LIN {X 0,Y 185.602,Z 322.354,A -85,B 0,C 180,E1 -22115.385,E2 -22115.385} C_VEL
LIN {X 0,Y 185.671,Z 322.353,A -85,B 0,C 180,E1 -22121.133,E2 -22121.133} C_VEL
LIN {X 0,Y 185.762,Z 322.338,A -85,B 0,C 180,E1 -22126.88,E2 -22126.88} C_VEL
LIN {X 0,Y 186.021,Z 322.304,A -85,B 0,C 180,E1 -22131.308,E2 -22131.308} C_VEL
LIN {X 0,Y 186.205,Z 322.287,A -85,B 0,C 180,E1 -22137.837,E2 -22137.837} C_VEL
LIN {X 0,Y 186.404,Z 322.255,A -85,B 0,C 180,E1 -22140.001,E2 -22140.001} C_VEL
LIN {X 0,Y 185.924,Z 322.314,A -85,B 0,C 180,E1 -22144.336,E2 -22144.336} C_VEL
LIN {X 0,Y 186.026,Z 322.301,A -85,B 0,C 180,E1 -22148.692,E2 -22148.692} C_VEL
LIN {X 0,Y 185.762,Z 322.334,A -85,B 0,C 180,E1 -22153.121,E2 -22153.121} C_VEL
LIN {X 0,Y 185.714,Z 322.341,A -85,B 0,C 180,E1 -22157.623,E2 -22157.623} C_VEL
LIN {X 0,Y 185.631,Z 322.481,A -85,B 0,C 180,E1 -22163.056,E2 -22163.056} C_VEL
LIN {X 0,Y 186.574,Z 325.065,A -85,B 0,C 180,E1 -22163.814,E2 -22163.814} C_VEL
LIN {X 0,Y 188.555,Z 327.314,A -85,B 0,C 180,E1 -22165.085,E2 -22165.085} C_VEL
LIN {X 0,Y 189.992,Z 328.26,A -85,B 0,C 180,E1 -22165.911,E2 -22165.911} C_VEL
LIN {X 0,Y 191.804,Z 331.332,A -85,B 0,C 180,E1 -22167.039,E2 -22167.039} C_VEL
LIN {X 0,Y 194.147,Z 333.688,A -85,B 0,C 180,E1 -22168.307,E2 -22168.307} C_VEL
LIN {X 0,Y 196.773,Z 337.354,A -85,B 0,C 180,E1 -22169.708,E2 -22169.708} C_VEL
LIN {X 0,Y 197.995,Z 338.775,A -85,B 0,C 180,E1 -22170.313,E2 -22170.313} C_VEL
LIN {X 0,Y 200.923,Z 342.622,A -85,B 0,C 180,E1 -22171.724,E2 -22171.724} C_VEL
LIN {X 0,Y 207.739,Z 352.452,A -85,B 0,C 180,E1 -22174.74,E2 -22174.74} C_VEL
LIN {X 0,Y 214.156,Z 362.539,A -85,B 0,C 180,E1 -22177.29,E2 -22177.29} C_VEL
LIN {X 0,Y 221.381,Z 375.322,A -85,B 0,C 180,E1 -22179.914,E2 -22179.914} C_VEL
LIN {X 0,Y 223.449,Z 379.739,A -85,B 0,C 180,E1 -22180.645,E2 -22180.645} C_VEL
LIN {X 0,Y 220.676,Z 423.154,A -85,B 0,C 180,E1 -22181.949,E2 -22181.949} C_VEL
LIN {X 0,Y 219.117,Z 436.689,A -85,B 0,C 180,E1 -22182.72,E2 -22182.72} C_VEL
LIN {X 0,Y 216.946,Z 448.789,A -85,B 0,C 180,E1 -22183.714,E2 -22183.714} C_VEL
LIN {X 0,Y 213.831,Z 460.908,A -85,B 0,C 180,E1 -22185.039,E2 -22185.039} C_VEL
LIN {X 0,Y 210.401,Z 472.488,A -85,B 0,C 180,E1 -22186.785,E2 -22186.785} C_VEL
LIN {X 0,Y 207.063,Z 482.377,A -85,B 0,C 180,E1 -22188.73,E2 -22188.73} C_VEL
LIN {X 0,Y 203.419,Z 491.299,A -85,B 0,C 180,E1 -22190.913,E2 -22190.913} C_VEL
LIN {X 0,Y 199.211,Z 500.425,A -85,B 0,C 180,E1 -22193.787,E2 -22193.787} C_VEL
LIN {X 0,Y 195.528,Z 507.705,A -85,B 0,C 180,E1 -22196.762,E2 -22196.762} C_VEL
LIN {X 0,Y 192.756,Z 512.596,A -85,B 0,C 180,E1 -22199.308,E2 -22199.308} C_VEL
LIN {X 0,Y 189.694,Z 517.737,A -85,B 0,C 180,E1 -22202.772,E2 -22202.772} C_VEL
LIN {X 0,Y 187.644,Z 520.887,A -85,B 0,C 180,E1 -22205.671,E2 -22205.671} C_VEL
LIN {X 0,Y 186.386,Z 522.696,A -85,B 0,C 180,E1 -22207.849,E2 -22207.849} C_VEL
LIN {X 0,Y 184.582,Z 524.972,A -85,B 0,C 180,E1 -22212.267,E2 -22212.267} C_VEL
LIN {X 0,Y 183.944,Z 525.517,A -85,B 0,C 180,E1 -22214.489,E2 -22214.489} C_VEL
LIN {X 0,Y 183.457,Z 525.636,A -85,B 0,C 180,E1 -22216.713,E2 -22216.713} C_VEL
LIN {X 0,Y 183.163,Z 524.659,A -85,B 0,C 180,E1 -22221.173,E2 -22221.173} C_VEL
LIN {X 0,Y 183.461,Z 522.612,A -85,B 0,C 180,E1 -22224.887,E2 -22224.887} C_VEL
LIN {X 0,Y 183.924,Z 519.046,A -85,B 0,C 180,E1 -22228.907,E2 -22228.907} C_VEL
LIN {X 0,Y 184.855,Z 514.96,A -85,B 0,C 180,E1 -22232.18,E2 -22232.18} C_VEL
LIN {X 0,Y 186.297,Z 508.724,A -85,B 0,C 180,E1 -22235.956,E2 -22235.956} C_VEL
LIN {X 0,Y 188.111,Z 501.932,A -85,B 0,C 180,E1 -22239.138,E2 -22239.138} C_VEL
LIN {X 0,Y 190.326,Z 493.47,A -85,B 0,C 180,E1 -22242.26,E2 -22242.26} C_VEL
LIN {X 0,Y 192.574,Z 484.767,A -85,B 0,C 180,E1 -22244.802,E2 -22244.802} C_VEL
LIN {X 0,Y 195.141,Z 474.056,A -85,B 0,C 180,E1 -22247.286,E2 -22247.286} C_VEL
LIN {X 0,Y 197.445,Z 463.339,A -85,B 0,C 180,E1 -22249.225,E2 -22249.225} C_VEL
LIN {X 0,Y 199.409,Z 451.373,A -85,B 0,C 180,E1 -22250.908,E2 -22250.908} C_VEL
LIN {X 0,Y 201.104,Z 438.875,A -85,B 0,C 180,E1 -22252.203,E2 -22252.203} C_VEL
LIN {X 0,Y 202.264,Z 426.146,A -85,B 0,C 180,E1 -22253.12,E2 -22253.12} C_VEL
LIN {X 0,Y 203.098,Z 410.38,A -85,B 0,C 180,E1 -22253.767,E2 -22253.767} C_VEL
LIN {X 0,Y 205.254,Z 361.08,A -85,B 0,C 180,E1 -22255.386,E2 -22255.386} C_VEL
LIN {X 0,Y 198.748,Z 346.766,A -85,B 0,C 180,E1 -22257.112,E2 -22257.112} C_VEL
LIN {X 0,Y 191.698,Z 333.496,A -85,B 0,C 180,E1 -22259.053,E2 -22259.053} C_VEL
LIN {X 0,Y 187.267,Z 326.204,A -85,B 0,C 180,E1 -22260.324,E2 -22260.324} C_VEL
LIN {X 0,Y 185.864,Z 323.755,A -85,B 0,C 180,E1 -22260.749,E2 -22260.749} C_VEL
LIN {X 0,Y 185.524,Z 322.374,A -85,B 0,C 180,E1 -22260.905,E2 -22260.905} C_VEL
LIN {X 0,Y 185.502,Z 322.377,A -85,B 0,C 180,E1 -22264.633,E2 -22264.633} C_VEL
LIN {X 0,Y 185.504,Z 322.377,A -85,B 0,C 180,E1 -22267.315,E2 -22267.315} C_VEL
LIN {X 0,Y 185.466,Z 322.369,A -85,B 0,C 180,E1 -22270.722,E2 -22270.722} C_VEL
LIN {X 0,Y 185.46,Z 322.373,A -85,B 0,C 180,E1 -22276.057,E2 -22276.057} C_VEL
LIN {X 0,Y 185.46,Z 322.377,A -85,B 0,C 180,E1 -22279.892,E2 -22279.892} C_VEL
LIN {X 0,Y 185.505,Z 322.374,A -85,B 0,C 180,E1 -22282.714,E2 -22282.714} C_VEL
LIN {X 0,Y 185.536,Z 322.367,A -85,B 0,C 180,E1 -22287.973,E2 -22287.973} C_VEL
LIN {X 0,Y 185.552,Z 322.371,A -85,B 0,C 180,E1 -22290.595,E2 -22290.595} C_VEL
LIN {X 0,Y 185.586,Z 322.342,A -85,B 0,C 180,E1 -22295.381,E2 -22295.381} C_VEL
LIN {X 0,Y 185.678,Z 322.353,A -85,B 0,C 180,E1 -22301.135,E2 -22301.135} C_VEL
LIN {X 0,Y 185.687,Z 322.326,A -85,B 0,C 180,E1 -22304.636,E2 -22304.636} C_VEL
LIN {X 0,Y 185.893,Z 322.327,A -85,B 0,C 180,E1 -22309.418,E2 -22309.418} C_VEL
LIN {X 0,Y 185.936,Z 322.305,A -85,B 0,C 180,E1 -22313.488,E2 -22313.488} C_VEL
LIN {X 0,Y 186.18,Z 322.28,A -85,B 0,C 180,E1 -22317.836,E2 -22317.836} C_VEL
LIN {X 0,Y 186.384,Z 322.266,A -85,B 0,C 180,E1 -22319.999,E2 -22319.999} C_VEL
LIN {X 0,Y 185.887,Z 322.311,A -85,B 0,C 180,E1 -22324.336,E2 -22324.336} C_VEL
LIN {X 0,Y 185.978,Z 322.305,A -85,B 0,C 180,E1 -22328.694,E2 -22328.694} C_VEL
LIN {X 0,Y 185.72,Z 322.346,A -85,B 0,C 180,E1 -22333.123,E2 -22333.123} C_VEL
LIN {X 0,Y 185.657,Z 322.356,A -85,B 0,C 180,E1 -22337.628,E2 -22337.628} C_VEL
LIN {X 0,Y 185.558,Z 322.37,A -85,B 0,C 180,E1 -22342.256,E2 -22342.256} C_VEL
LIN {X 0,Y 185.581,Z 322.37,A -85,B 0,C 180,E1 -22344.645,E2 -22344.645} C_VEL
LIN {X 0,Y 185.547,Z 322.374,A -85,B 0,C 180,E1 -22349.498,E2 -22349.498} C_VEL
LIN {X 0,Y 185.5,Z 322.381,A -85,B 0,C 180,E1 -22354.632,E2 -22354.632} C_VEL
LIN {X 0,Y 185.502,Z 322.38,A -85,B 0,C 180,E1 -22357.313,E2 -22357.313} C_VEL
LIN {X 0,Y 185.464,Z 322.384,A -85,B 0,C 180,E1 -22360.72,E2 -22360.72} C_VEL
LIN {X 0,Y 185.457,Z 322.381,A -85,B 0,C 180,E1 -22366.055,E2 -22366.055} C_VEL
LIN {X 0,Y 185.455,Z 322.498,A -85,B 0,C 180,E1 -22366.666,E2 -22366.666} C_VEL
LIN {X 0,Y 187.234,Z 328.959,A -85,B 0,C 180,E1 -22370.164,E2 -22370.164} C_VEL
LIN {X 0,Y 193.7,Z 342.579,A -85,B 0,C 180,E1 -22372.115,E2 -22372.115} C_VEL
LIN {X 0,Y 199.635,Z 357.226,A -85,B 0,C 180,E1 -22373.852,E2 -22373.852} C_VEL
LIN {X 0,Y 201.477,Z 362.857,A -85,B 0,C 180,E1 -22374.409,E2 -22374.409} C_VEL
LIN {X 0,Y 203.893,Z 387.642,A -85,B 0,C 180,E1 -22375.818,E2 -22375.818} C_VEL
LIN {X 0,Y 204.068,Z 393.676,A -85,B 0,C 180,E1 -22376.087,E2 -22376.087} C_VEL
LIN {X 0,Y 203.042,Z 418.397,A -85,B 0,C 180,E1 -22376.909,E2 -22376.909} C_VEL
LIN {X 0,Y 202.212,Z 424.252,A -85,B 0,C 180,E1 -22377.003,E2 -22377.003} C_VEL
LIN {X 0,Y 196.642,Z 441.249,A -85,B 0,C 180,E1 -22376.926,E2 -22376.926} C_VEL
LIN {X 0,Y 195.203,Z 446.94,A -85,B 0,C 180,E1 -22377.129,E2 -22377.129} C_VEL
LIN {X 0,Y 194.917,Z 448.84,A -85,B 0,C 180,E1 -22377.257,E2 -22377.257} C_VEL
LIN {X 0,Y 192.992,Z 462.243,A -85,B 0,C 180,E1 -22378.432,E2 -22378.432} C_VEL
LIN {X 0,Y 190.833,Z 474.025,A -85,B 0,C 180,E1 -22379.881,E2 -22379.881} C_VEL
LIN {X 0,Y 188.453,Z 484.745,A -85,B 0,C 180,E1 -22381.607,E2 -22381.607} C_VEL
LIN {X 0,Y 185.81,Z 495.707,A -85,B 0,C 180,E1 -22383.914,E2 -22383.914} C_VEL
LIN {X 0,Y 183.52,Z 504.648,A -85,B 0,C 180,E1 -22386.289,E2 -22386.289} C_VEL
LIN {X 0,Y 181.358,Z 512.767,A -85,B 0,C 180,E1 -22388.957,E2 -22388.957} C_VEL
LIN {X 0,Y 179.325,Z 520.919,A -85,B 0,C 180,E1 -22392.317,E2 -22392.317} C_VEL
LIN {X 0,Y 177.916,Z 526.35,A -85,B 0,C 180,E1 -22395.121,E2 -22395.121} C_VEL
LIN {X 0,Y 176.864,Z 531.673,A -85,B 0,C 180,E1 -22398.539,E2 -22398.539} C_VEL
LIN {X 0,Y 176.312,Z 535.798,A -85,B 0,C 180,E1 -22401.979,E2 -22401.979} C_VEL
LIN {X 0,Y 176.155,Z 539.184,A -85,B 0,C 180,E1 -22405.88,E2 -22405.88} C_VEL
LIN {X 0,Y 176.344,Z 541.364,A -85,B 0,C 180,E1 -22409.999,E2 -22409.999} C_VEL
LIN {X 0,Y 176.067,Z 542.161,A -85,B 0,C 180,E1 -22413.703,E2 -22413.703} C_VEL
LIN {X 0,Y 176.127,Z 542.036,A -85,B 0,C 180,E1 -22416.874,E2 -22416.874} C_VEL
LIN {X 0,Y 176.941,Z 540.465,A -85,B 0,C 180,E1 -22421.453,E2 -22421.453} C_VEL
LIN {X 0,Y 178.663,Z 537.326,A -85,B 0,C 180,E1 -22425.982,E2 -22425.982} C_VEL
LIN {X 0,Y 180.848,Z 533.822,A -85,B 0,C 180,E1 -22429.287,E2 -22429.287} C_VEL
LIN {X 0,Y 183.561,Z 529.251,A -85,B 0,C 180,E1 -22432.51,E2 -22432.51} C_VEL
LIN {X 0,Y 187.209,Z 522.474,A -85,B 0,C 180,E1 -22436.113,E2 -22436.113} C_VEL
LIN {X 0,Y 191.164,Z 514.93,A -85,B 0,C 180,E1 -22439.15,E2 -22439.15} C_VEL
LIN {X 0,Y 195.701,Z 505.709,A -85,B 0,C 180,E1 -22441.984,E2 -22441.984} C_VEL
LIN {X 0,Y 200.276,Z 495.091,A -85,B 0,C 180,E1 -22444.46,E2 -22444.46} C_VEL
LIN {X 0,Y 204.387,Z 484.289,A -85,B 0,C 180,E1 -22446.379,E2 -22446.379} C_VEL
LIN {X 0,Y 207.698,Z 473.768,A -85,B 0,C 180,E1 -22447.827,E2 -22447.827} C_VEL
LIN {X 0,Y 210.983,Z 461.115,A -85,B 0,C 180,E1 -22449.109,E2 -22449.109} C_VEL
LIN {X 0,Y 213.479,Z 448.246,A -85,B 0,C 180,E1 -22450.038,E2 -22450.038} C_VEL
LIN {X 0,Y 214.982,Z 435.79,A -85,B 0,C 180,E1 -22450.639,E2 -22450.639} C_VEL
LIN {X 0,Y 217.345,Z 398.415,A -85,B 0,C 180,E1 -22451.778,E2 -22451.778} C_VEL
LIN {X 0,Y 216.378,Z 390.526,A -85,B 0,C 180,E1 -22452.408,E2 -22452.408} C_VEL
LIN {X 0,Y 211.348,Z 378.41,A -85,B 0,C 180,E1 -22454.445,E2 -22454.445} C_VEL
LIN {X 0,Y 206.149,Z 367.504,A -85,B 0,C 180,E1 -22456.668,E2 -22456.668} C_VEL
LIN {X 0,Y 200.479,Z 357.126,A -85,B 0,C 180,E1 -22459.272,E2 -22459.272} C_VEL
LIN {X 0,Y 195.398,Z 348.706,A -85,B 0,C 180,E1 -22461.837,E2 -22461.837} C_VEL
LIN {X 0,Y 192.188,Z 343.632,A -85,B 0,C 180,E1 -22463.607,E2 -22463.607} C_VEL
LIN {X 0,Y 189.031,Z 338.725,A -85,B 0,C 180,E1 -22465.496,E2 -22465.496} C_VEL
LIN {X 0,Y 184.565,Z 332.55,A -85,B 0,C 180,E1 -22468.428,E2 -22468.428} C_VEL
LIN {X 0,Y 183.865,Z 331.486,A -85,B 0,C 180,E1 -22468.935,E2 -22468.935} C_VEL
LIN {X 0,Y 180.936,Z 328.003,A -85,B 0,C 180,E1 -22471.123,E2 -22471.123} C_VEL
LIN {X 0,Y 178.979,Z 324.987,A -85,B 0,C 180,E1 -22472.84,E2 -22472.84} C_VEL
LIN {X 0,Y 178.558,Z 323.232,A -85,B 0,C 180,E1 -22475.114,E2 -22475.114} C_VEL
LIN {X 0,Y 178.65,Z 323.232,A -85,B 0,C 180,E1 -22481.657,E2 -22481.657} C_VEL
LIN {X 0,Y 178.679,Z 323.224,A -85,B 0,C 180,E1 -22486.35,E2 -22486.35} C_VEL
LIN {X 0,Y 178.971,Z 323.184,A -85,B 0,C 180,E1 -22490.963,E2 -22490.963} C_VEL
LIN {X 0,Y 179.151,Z 323.164,A -85,B 0,C 180,E1 -22497.752,E2 -22497.752} C_VEL
LIN {X 0,Y 179.367,Z 323.131,A -85,B 0,C 180,E1 -22500.001,E2 -22500.001} C_VEL
LIN {X 0,Y 178.872,Z 323.192,A -85,B 0,C 180,E1 -22504.508,E2 -22504.508} C_VEL
LIN {X 0,Y 178.975,Z 323.179,A -85,B 0,C 180,E1 -22509.038,E2 -22509.038} C_VEL
LIN {X 0,Y 178.686,Z 323.215,A -85,B 0,C 180,E1 -22513.651,E2 -22513.651} C_VEL
LIN {X 0,Y 178.685,Z 323.334,A -85,B 0,C 180,E1 -22518.489,E2 -22518.489} C_VEL
LIN {X 0,Y 179.446,Z 325.802,A -85,B 0,C 180,E1 -22519.299,E2 -22519.299} C_VEL
LIN {X 0,Y 181.37,Z 328.083,A -85,B 0,C 180,E1 -22520.856,E2 -22520.856} C_VEL
LIN {X 0,Y 183.347,Z 329.344,A -85,B 0,C 180,E1 -22522.243,E2 -22522.243} C_VEL
LIN {X 0,Y 185.208,Z 332.563,A -85,B 0,C 180,E1 -22523.629,E2 -22523.629} C_VEL
LIN {X 0,Y 187.704,Z 334.907,A -85,B 0,C 180,E1 -22525.207,E2 -22525.207} C_VEL
LIN {X 0,Y 190.012,Z 338.227,A -85,B 0,C 180,E1 -22526.646,E2 -22526.646} C_VEL
LIN {X 0,Y 191.662,Z 340.012,A -85,B 0,C 180,E1 -22527.578,E2 -22527.578} C_VEL
LIN {X 0,Y 194.472,Z 343.763,A -85,B 0,C 180,E1 -22529.12,E2 -22529.12} C_VEL
LIN {X 0,Y 200.952,Z 352.705,A -85,B 0,C 180,E1 -22532.33,E2 -22532.33} C_VEL
LIN {X 0,Y 206.555,Z 361.344,A -85,B 0,C 180,E1 -22534.819,E2 -22534.819} C_VEL
LIN {X 0,Y 212.088,Z 370.486,A -85,B 0,C 180,E1 -22537.063,E2 -22537.063} C_VEL
LIN {X 0,Y 218.186,Z 381.915,A -85,B 0,C 180,E1 -22539.365,E2 -22539.365} C_VEL
LIN {X 0,Y 218.038,Z 386.773,A -85,B 0,C 180,E1 -22539.55,E2 -22539.55} C_VEL
LIN {X 0,Y 215.55,Z 423.517,A -85,B 0,C 180,E1 -22540.666,E2 -22540.666} C_VEL
LIN {X 0,Y 213.893,Z 437.147,A -85,B 0,C 180,E1 -22541.449,E2 -22541.449} C_VEL
LIN {X 0,Y 211.532,Z 449.75,A -85,B 0,C 180,E1 -22542.511,E2 -22542.511} C_VEL
LIN {X 0,Y 208.303,Z 461.709,A -85,B 0,C 180,E1 -22543.85,E2 -22543.85} C_VEL
LIN {X 0,Y 204.738,Z 473.203,A -85,B 0,C 180,E1 -22545.622,E2 -22545.622} C_VEL
LIN {X 0,Y 201.485,Z 482.435,A -85,B 0,C 180,E1 -22547.477,E2 -22547.477} C_VEL
LIN {X 0,Y 197.837,Z 491.031,A -85,B 0,C 180,E1 -22549.587,E2 -22549.587} C_VEL
LIN {X 0,Y 194.137,Z 498.886,A -85,B 0,C 180,E1 -22552.019,E2 -22552.019} C_VEL
LIN {X 0,Y 190.113,Z 506.513,A -85,B 0,C 180,E1 -22555.042,E2 -22555.042} C_VEL
LIN {X 0,Y 186.545,Z 512.606,A -85,B 0,C 180,E1 -22558.169,E2 -22558.169} C_VEL
LIN {X 0,Y 183.485,Z 517.458,A -85,B 0,C 180,E1 -22561.451,E2 -22561.451} C_VEL
LIN {X 0,Y 181.037,Z 521.031,A -85,B 0,C 180,E1 -22564.722,E2 -22564.722} C_VEL
LIN {X 0,Y 179.685,Z 522.891,A -85,B 0,C 180,E1 -22566.977,E2 -22566.977} C_VEL
LIN {X 0,Y 178.576,Z 524.269,A -85,B 0,C 180,E1 -22569.257,E2 -22569.257} C_VEL
LIN {X 0,Y 177.621,Z 525.297,A -85,B 0,C 180,E1 -22571.738,E2 -22571.738} C_VEL
LIN {X 0,Y 176.466,Z 525.982,A -85,B 0,C 180,E1 -22576.176,E2 -22576.176} C_VEL
LIN {X 0,Y 176.059,Z 525.066,A -85,B 0,C 180,E1 -22580.814,E2 -22580.814} C_VEL
LIN {X 0,Y 176.381,Z 522.887,A -85,B 0,C 180,E1 -22584.974,E2 -22584.974} C_VEL
LIN {X 0,Y 176.833,Z 519.596,A -85,B 0,C 180,E1 -22588.863,E2 -22588.863} C_VEL
LIN {X 0,Y 177.763,Z 515.576,A -85,B 0,C 180,E1 -22592.267,E2 -22592.267} C_VEL
LIN {X 0,Y 179.267,Z 509.413,A -85,B 0,C 180,E1 -22596.191,E2 -22596.191} C_VEL
LIN {X 0,Y 181.109,Z 502.703,A -85,B 0,C 180,E1 -22599.494,E2 -22599.494} C_VEL
LIN {X 0,Y 183.419,Z 494.376,A -85,B 0,C 180,E1 -22602.729,E2 -22602.729} C_VEL
LIN {X 0,Y 185.75,Z 485.791,A -85,B 0,C 180,E1 -22605.36,E2 -22605.36} C_VEL
LIN {X 0,Y 188.43,Z 475.216,A -85,B 0,C 180,E1 -22607.922,E2 -22607.922} C_VEL
LIN {X 0,Y 190.803,Z 464.712,A -85,B 0,C 180,E1 -22609.922,E2 -22609.922} C_VEL
LIN {X 0,Y 192.865,Z 453.102,A -85,B 0,C 180,E1 -22611.653,E2 -22611.653} C_VEL
LIN {X 0,Y 194.603,Z 441.042,A -85,B 0,C 180,E1 -22612.986,E2 -22612.986} C_VEL
LIN {X 0,Y 195.932,Z 427.802,A -85,B 0,C 180,E1 -22614.021,E2 -22614.021} C_VEL
LIN {X 0,Y 196.763,Z 414.296,A -85,B 0,C 180,E1 -22614.639,E2 -22614.639} C_VEL
LIN {X 0,Y 199.121,Z 362.92,A -85,B 0,C 180,E1 -22616.367,E2 -22616.367} C_VEL
LIN {X 0,Y 192.412,Z 348.456,A -85,B 0,C 180,E1 -22618.246,E2 -22618.246} C_VEL
LIN {X 0,Y 186.566,Z 337.49,A -85,B 0,C 180,E1 -22619.953,E2 -22619.953} C_VEL
LIN {X 0,Y 180.371,Z 327.254,A -85,B 0,C 180,E1 -22621.859,E2 -22621.859} C_VEL
LIN {X 0,Y 178.84,Z 324.725,A -85,B 0,C 180,E1 -22622.358,E2 -22622.358} C_VEL
LIN {X 0,Y 178.498,Z 323.25,A -85,B 0,C 180,E1 -22622.599,E2 -22622.599} C_VEL
LIN {X 0,Y 178.411,Z 323.261,A -85,B 0,C 180,E1 -22628.014,E2 -22628.014} C_VEL
LIN {X 0,Y 178.398,Z 323.251,A -85,B 0,C 180,E1 -22632.047,E2 -22632.047} C_VEL
LIN {X 0,Y 178.396,Z 323.258,A -85,B 0,C 180,E1 -22635.165,E2 -22635.165} C_VEL
LIN {X 0,Y 178.401,Z 323.245,A -85,B 0,C 180,E1 -22638.462,E2 -22638.462} C_VEL
LIN {X 0,Y 178.423,Z 323.246,A -85,B 0,C 180,E1 -22643.782,E2 -22643.782} C_VEL
LIN {X 0,Y 178.489,Z 323.233,A -85,B 0,C 180,E1 -22646.546,E2 -22646.546} C_VEL
LIN {X 0,Y 178.447,Z 323.25,A -85,B 0,C 180,E1 -22651.795,E2 -22651.795} C_VEL
LIN {X 0,Y 178.52,Z 323.22,A -85,B 0,C 180,E1 -22654.889,E2 -22654.889} C_VEL
LIN {X 0,Y 178.626,Z 323.232,A -85,B 0,C 180,E1 -22660.787,E2 -22660.787} C_VEL
LIN {X 0,Y 178.654,Z 323.208,A -85,B 0,C 180,E1 -22666.347,E2 -22666.347} C_VEL
LIN {X 0,Y 178.911,Z 323.196,A -85,B 0,C 180,E1 -22670.959,E2 -22670.959} C_VEL
LIN {X 0,Y 179.128,Z 323.157,A -85,B 0,C 180,E1 -22677.751,E2 -22677.751} C_VEL
LIN {X 0,Y 179.349,Z 323.142,A -85,B 0,C 180,E1 -22679.999,E2 -22679.999} C_VEL
LIN {X 0,Y 178.836,Z 323.187,A -85,B 0,C 180,E1 -22684.507,E2 -22684.507} C_VEL
LIN {X 0,Y 178.909,Z 323.188,A -85,B 0,C 180,E1 -22689.04,E2 -22689.04} C_VEL
LIN {X 0,Y 178.647,Z 323.227,A -85,B 0,C 180,E1 -22693.652,E2 -22693.652} C_VEL
LIN {X 0,Y 178.558,Z 323.241,A -85,B 0,C 180,E1 -22699.151,E2 -22699.151} C_VEL
LIN {X 0,Y 178.519,Z 323.251,A -85,B 0,C 180,E1 -22705.11,E2 -22705.11} C_VEL
LIN {X 0,Y 178.463,Z 323.254,A -85,B 0,C 180,E1 -22710.793,E2 -22710.793} C_VEL
LIN {X 0,Y 178.485,Z 323.254,A -85,B 0,C 180,E1 -22714.217,E2 -22714.217} C_VEL
LIN {X 0,Y 178.39,Z 323.266,A -85,B 0,C 180,E1 -22719.076,E2 -22719.076} C_VEL
LIN {X 0,Y 178.396,Z 323.264,A -85,B 0,C 180,E1 -22722.045,E2 -22722.045} C_VEL
LIN {X 0,Y 178.404,Z 323.332,A -85,B 0,C 180,E1 -22725.461,E2 -22725.461} C_VEL
LIN {X 0,Y 179.755,Z 328.364,A -85,B 0,C 180,E1 -22728.414,E2 -22728.414} C_VEL
LIN {X 0,Y 186.912,Z 342.847,A -85,B 0,C 180,E1 -22730.735,E2 -22730.735} C_VEL
LIN {X 0,Y 192.782,Z 356.972,A -85,B 0,C 180,E1 -22732.565,E2 -22732.565} C_VEL
LIN {X 0,Y 195.565,Z 365.01,A -85,B 0,C 180,E1 -22733.441,E2 -22733.441} C_VEL
LIN {X 0,Y 197.964,Z 390.894,A -85,B 0,C 180,E1 -22734.959,E2 -22734.959} C_VEL
LIN {X 0,Y 195.933,Z 438.172,A -85,B 0,C 180,E1 -22736.635,E2 -22736.635} C_VEL
LIN {X 0,Y 194.917,Z 448.84,A -85,B 0,C 180,E1 -22737.257,E2 -22737.257} C_VEL
LIN {X 0,Y 194.124,Z 452.609,A -85,B 0,C 180,E1 -22737.495,E2 -22737.495} C_VEL
LIN {X 0,Y 191.322,Z 459.899,A -85,B 0,C 180,E1 -22737.876,E2 -22737.876} C_VEL
LIN {X 0,Y 186.171,Z 470.409,A -85,B 0,C 180,E1 -22738.6,E2 -22738.6} C_VEL
LIN {X 0,Y 184.192,Z 475.629,A -85,B 0,C 180,E1 -22739.215,E2 -22739.215} C_VEL
LIN {X 0,Y 183.741,Z 477.33,A -85,B 0,C 180,E1 -22739.473,E2 -22739.473} C_VEL
LIN {X 0,Y 180.934,Z 488.925,A -85,B 0,C 180,E1 -22741.585,E2 -22741.585} C_VEL
LIN {X 0,Y 178.576,Z 498.019,A -85,B 0,C 180,E1 -22743.719,E2 -22743.719} C_VEL
LIN {X 0,Y 175.998,Z 507.339,A -85,B 0,C 180,E1 -22746.463,E2 -22746.463} C_VEL
LIN {X 0,Y 174.317,Z 513.626,A -85,B 0,C 180,E1 -22748.723,E2 -22748.723} C_VEL
LIN {X 0,Y 172.196,Z 521.426,A -85,B 0,C 180,E1 -22752.174,E2 -22752.174} C_VEL
LIN {X 0,Y 170.521,Z 527.665,A -85,B 0,C 180,E1 -22755.681,E2 -22755.681} C_VEL
LIN {X 0,Y 169.62,Z 532.628,A -85,B 0,C 180,E1 -22759.253,E2 -22759.253} C_VEL
LIN {X 0,Y 169.147,Z 536.434,A -85,B 0,C 180,E1 -22762.838,E2 -22762.838} C_VEL
LIN {X 0,Y 169.074,Z 538.963,A -85,B 0,C 180,E1 -22766.046,E2 -22766.046} C_VEL
LIN {X 0,Y 169.26,Z 540.98,A -85,B 0,C 180,E1 -22769.998,E2 -22769.998} C_VEL
LIN {X 0,Y 168.986,Z 541.801,A -85,B 0,C 180,E1 -22773.495,E2 -22773.495} C_VEL
LIN {X 0,Y 169.078,Z 541.727,A -85,B 0,C 180,E1 -22777.162,E2 -22777.162} C_VEL
LIN {X 0,Y 169.967,Z 540.211,A -85,B 0,C 180,E1 -22781.93,E2 -22781.93} C_VEL
LIN {X 0,Y 171.829,Z 537.127,A -85,B 0,C 180,E1 -22786.635,E2 -22786.635} C_VEL
LIN {X 0,Y 174.143,Z 533.665,A -85,B 0,C 180,E1 -22790.061,E2 -22790.061} C_VEL
LIN {X 0,Y 177.665,Z 528.009,A -85,B 0,C 180,E1 -22794.099,E2 -22794.099} C_VEL
LIN {X 0,Y 181.532,Z 521.22,A -85,B 0,C 180,E1 -22797.681,E2 -22797.681} C_VEL
LIN {X 0,Y 185.754,Z 513.615,A -85,B 0,C 180,E1 -22800.714,E2 -22800.714} C_VEL
LIN {X 0,Y 189.725,Z 505.861,A -85,B 0,C 180,E1 -22803.118,E2 -22803.118} C_VEL
LIN {X 0,Y 194.483,Z 495.352,A -85,B 0,C 180,E1 -22805.639,E2 -22805.639} C_VEL
LIN {X 0,Y 198.715,Z 484.68,A -85,B 0,C 180,E1 -22807.594,E2 -22807.594} C_VEL
LIN {X 0,Y 202.164,Z 474.367,A -85,B 0,C 180,E1 -22809.055,E2 -22809.055} C_VEL
LIN {X 0,Y 205.558,Z 462.032,A -85,B 0,C 180,E1 -22810.349,E2 -22810.349} C_VEL
LIN {X 0,Y 208.311,Z 448.604,A -85,B 0,C 180,E1 -22811.348,E2 -22811.348} C_VEL
LIN {X 0,Y 209.889,Z 436.585,A -85,B 0,C 180,E1 -22811.957,E2 -22811.957} C_VEL
LIN {X 0,Y 212.359,Z 399.603,A -85,B 0,C 180,E1 -22813.101,E2 -22813.101} C_VEL
LIN {X 0,Y 211.595,Z 393.444,A -85,B 0,C 180,E1 -22813.625,E2 -22813.625} C_VEL
LIN {X 0,Y 206.667,Z 381.356,A -85,B 0,C 180,E1 -22815.76,E2 -22815.76} C_VEL
LIN {X 0,Y 201.226,Z 369.955,A -85,B 0,C 180,E1 -22818.253,E2 -22818.253} C_VEL
LIN {X 0,Y 195.946,Z 360.193,A -85,B 0,C 180,E1 -22820.881,E2 -22820.881} C_VEL
LIN {X 0,Y 191.874,Z 353.48,A -85,B 0,C 180,E1 -22823.085,E2 -22823.085} C_VEL
LIN {X 0,Y 189.122,Z 349.043,A -85,B 0,C 180,E1 -22824.701,E2 -22824.701} C_VEL
LIN {X 0,Y 185.725,Z 343.763,A -85,B 0,C 180,E1 -22826.869,E2 -22826.869} C_VEL
LIN {X 0,Y 181.515,Z 337.607,A -85,B 0,C 180,E1 -22829.877,E2 -22829.877} C_VEL
LIN {X 0,Y 177.174,Z 331.692,A -85,B 0,C 180,E1 -22833.497,E2 -22833.497} C_VEL
LIN {X 0,Y 175.105,Z 329.437,A -85,B 0,C 180,E1 -22835.443,E2 -22835.443} C_VEL
LIN {X 0,Y 172.644,Z 327.27,A -85,B 0,C 180,E1 -22838.038,E2 -22838.038} C_VEL
LIN {X 0,Y 171.706,Z 325.099,A -85,B 0,C 180,E1 -22839.344,E2 -22839.344} C_VEL
LIN {X 0,Y 171.522,Z 324.107,A -85,B 0,C 180,E1 -22839.762,E2 -22839.762} C_VEL
LIN {X 0,Y 171.557,Z 324.105,A -85,B 0,C 180,E1 -22843.336,E2 -22843.336} C_VEL
LIN {X 0,Y 171.846,Z 324.072,A -85,B 0,C 180,E1 -22848.963,E2 -22848.963} C_VEL
LIN {X 0,Y 171.893,Z 324.064,A -85,B 0,C 180,E1 -22852.955,E2 -22852.955} C_VEL
LIN {X 0,Y 172.099,Z 324.041,A -85,B 0,C 180,E1 -22857.66,E2 -22857.66} C_VEL
LIN {X 0,Y 172.33,Z 324.007,A -85,B 0,C 180,E1 -22860.001,E2 -22860.001} C_VEL
LIN {X 0,Y 171.822,Z 324.069,A -85,B 0,C 180,E1 -22864.693,E2 -22864.693} C_VEL
LIN {X 0,Y 171.907,Z 324.059,A -85,B 0,C 180,E1 -22869.413,E2 -22869.413} C_VEL
LIN {X 0,Y 171.711,Z 324.089,A -85,B 0,C 180,E1 -22872.184,E2 -22872.184} C_VEL
LIN {X 0,Y 172.277,Z 326.189,A -85,B 0,C 180,E1 -22873.117,E2 -22873.117} C_VEL
LIN {X 0,Y 173.806,Z 328.419,A -85,B 0,C 180,E1 -22874.939,E2 -22874.939} C_VEL
LIN {X 0,Y 176.69,Z 330.308,A -85,B 0,C 180,E1 -22877.656,E2 -22877.656} C_VEL
LIN {X 0,Y 178.22,Z 333.282,A -85,B 0,C 180,E1 -22879.135,E2 -22879.135} C_VEL
LIN {X 0,Y 180.715,Z 335.426,A -85,B 0,C 180,E1 -22881.084,E2 -22881.084} C_VEL
LIN {X 0,Y 181.353,Z 336.116,A -85,B 0,C 180,E1 -22881.565,E2 -22881.565} C_VEL
LIN {X 0,Y 183.477,Z 339.361,A -85,B 0,C 180,E1 -22883.165,E2 -22883.165} C_VEL
LIN {X 0,Y 185.378,Z 341.21,A -85,B 0,C 180,E1 -22884.416,E2 -22884.416} C_VEL
LIN {X 0,Y 188.037,Z 344.866,A -85,B 0,C 180,E1 -22886.126,E2 -22886.126} C_VEL
LIN {X 0,Y 189.327,Z 346.504,A -85,B 0,C 180,E1 -22886.899,E2 -22886.899} C_VEL
LIN {X 0,Y 193.428,Z 352.176,A -85,B 0,C 180,E1 -22889.21,E2 -22889.21} C_VEL
LIN {X 0,Y 197.946,Z 358.508,A -85,B 0,C 180,E1 -22891.507,E2 -22891.507} C_VEL
LIN {X 0,Y 203.63,Z 367.481,A -85,B 0,C 180,E1 -22894.149,E2 -22894.149} C_VEL
LIN {X 0,Y 209.859,Z 378.252,A -85,B 0,C 180,E1 -22896.772,E2 -22896.772} C_VEL
LIN {X 0,Y 213.207,Z 384.749,A -85,B 0,C 180,E1 -22898.101,E2 -22898.101} C_VEL
LIN {X 0,Y 210.55,Z 423.817,A -85,B 0,C 180,E1 -22899.32,E2 -22899.32} C_VEL
LIN {X 0,Y 208.796,Z 437.62,A -85,B 0,C 180,E1 -22900.121,E2 -22900.121} C_VEL
LIN {X 0,Y 206.471,Z 449.646,A -85,B 0,C 180,E1 -22901.142,E2 -22901.142} C_VEL
LIN {X 0,Y 203.385,Z 460.908,A -85,B 0,C 180,E1 -22902.388,E2 -22902.388} C_VEL
LIN {X 0,Y 199.599,Z 472.604,A -85,B 0,C 180,E1 -22904.16,E2 -22904.16} C_VEL
LIN {X 0,Y 196,Z 482.504,A -85,B 0,C 180,E1 -22906.155,E2 -22906.155} C_VEL
LIN {X 0,Y 191.559,Z 492.444,A -85,B 0,C 180,E1 -22908.672,E2 -22908.672} C_VEL
LIN {X 0,Y 186.96,Z 501.471,A -85,B 0,C 180,E1 -22911.667,E2 -22911.667} C_VEL
LIN {X 0,Y 182.908,Z 508.688,A -85,B 0,C 180,E1 -22914.807,E2 -22914.807} C_VEL
LIN {X 0,Y 179.269,Z 514.388,A -85,B 0,C 180,E1 -22918.047,E2 -22918.047} C_VEL
LIN {X 0,Y 176.234,Z 518.84,A -85,B 0,C 180,E1 -22921.411,E2 -22921.411} C_VEL
LIN {X 0,Y 174.507,Z 521.175,A -85,B 0,C 180,E1 -22923.706,E2 -22923.706} C_VEL
LIN {X 0,Y 173.017,Z 523.07,A -85,B 0,C 180,E1 -22926.035,E2 -22926.035} C_VEL
LIN {X 0,Y 171.816,Z 524.505,A -85,B 0,C 180,E1 -22928.401,E2 -22928.401} C_VEL
LIN {X 0,Y 170.052,Z 526.102,A -85,B 0,C 180,E1 -22933.185,E2 -22933.185} C_VEL
LIN {X 0,Y 169.493,Z 526.315,A -85,B 0,C 180,E1 -22935.596,E2 -22935.596} C_VEL
LIN {X 0,Y 169.103,Z 526.096,A -85,B 0,C 180,E1 -22938.008,E2 -22938.008} C_VEL
LIN {X 0,Y 169.081,Z 524.457,A -85,B 0,C 180,E1 -22942.838,E2 -22942.838} C_VEL
LIN {X 0,Y 169.299,Z 523.051,A -85,B 0,C 180,E1 -22945.239,E2 -22945.239} C_VEL
LIN {X 0,Y 169.743,Z 520.125,A -85,B 0,C 180,E1 -22948.815,E2 -22948.815} C_VEL
LIN {X 0,Y 170.654,Z 516.17,A -85,B 0,C 180,E1 -22952.362,E2 -22952.362} C_VEL
LIN {X 0,Y 171.992,Z 511.087,A -85,B 0,C 180,E1 -22955.865,E2 -22955.865} C_VEL
LIN {X 0,Y 173.767,Z 504.693,A -85,B 0,C 180,E1 -22959.312,E2 -22959.312} C_VEL
LIN {X 0,Y 176.093,Z 496.721,A -85,B 0,C 180,E1 -22962.682,E2 -22962.682} C_VEL
LIN {X 0,Y 178.451,Z 488.59,A -85,B 0,C 180,E1 -22965.418,E2 -22965.418} C_VEL
LIN {X 0,Y 181.152,Z 478.675,A -85,B 0,C 180,E1 -22968.083,E2 -22968.083} C_VEL
LIN {X 0,Y 183.854,Z 467.465,A -85,B 0,C 180,E1 -22970.416,E2 -22970.416} C_VEL
LIN {X 0,Y 186.044,Z 456.512,A -85,B 0,C 180,E1 -22972.196,E2 -22972.196} C_VEL
LIN {X 0,Y 187.948,Z 444.407,A -85,B 0,C 180,E1 -22973.703,E2 -22973.703} C_VEL
LIN {X 0,Y 189.487,Z 431.517,A -85,B 0,C 180,E1 -22974.825,E2 -22974.825} C_VEL
LIN {X 0,Y 190.427,Z 418.197,A -85,B 0,C 180,E1 -22975.564,E2 -22975.564} C_VEL
LIN {X 0,Y 193.037,Z 364.96,A -85,B 0,C 180,E1 -22977.402,E2 -22977.402} C_VEL
LIN {X 0,Y 186.938,Z 351.779,A -85,B 0,C 180,E1 -22979.215,E2 -22979.215} C_VEL
LIN {X 0,Y 181.331,Z 341.27,A -85,B 0,C 180,E1 -22980.949,E2 -22980.949} C_VEL
LIN {X 0,Y 175.237,Z 331.189,A -85,B 0,C 180,E1 -22982.94,E2 -22982.94} C_VEL
LIN {X 0,Y 173.444,Z 328.239,A -85,B 0,C 180,E1 -22983.562,E2 -22983.562} C_VEL
LIN {X 0,Y 171.86,Z 325.8,A -85,B 0,C 180,E1 -22984.117,E2 -22984.117} C_VEL
LIN {X 0,Y 171.441,Z 324.129,A -85,B 0,C 180,E1 -22984.375,E2 -22984.375} C_VEL
LIN {X 0,Y 171.347,Z 324.14,A -85,B 0,C 180,E1 -22988.802,E2 -22988.802} C_VEL
LIN {X 0,Y 171.323,Z 324.142,A -85,B 0,C 180,E1 -22994.219,E2 -22994.219} C_VEL
LIN {X 0,Y 171.334,Z 324.128,A -85,B 0,C 180,E1 -22998.98,E2 -22998.98} C_VEL
LIN {X 0,Y 171.364,Z 324.136,A -85,B 0,C 180,E1 -23002.034,E2 -23002.034} C_VEL
LIN {X 0,Y 171.402,Z 324.111,A -85,B 0,C 180,E1 -23005.093,E2 -23005.093} C_VEL
LIN {X 0,Y 171.413,Z 324.132,A -85,B 0,C 180,E1 -23010.527,E2 -23010.527} C_VEL
LIN {X 0,Y 171.445,Z 324.104,A -85,B 0,C 180,E1 -23015.799,E2 -23015.799} C_VEL
LIN {X 0,Y 171.582,Z 324.109,A -85,B 0,C 180,E1 -23020.871,E2 -23020.871} C_VEL
LIN {X 0,Y 171.571,Z 324.085,A -85,B 0,C 180,E1 -23025.772,E2 -23025.772} C_VEL
LIN {X 0,Y 171.849,Z 324.077,A -85,B 0,C 180,E1 -23030.584,E2 -23030.584} C_VEL
LIN {X 0,Y 171.787,Z 324.053,A -85,B 0,C 180,E1 -23035.306,E2 -23035.306} C_VEL
LIN {X 0,Y 172.314,Z 324.018,A -85,B 0,C 180,E1 -23039.999,E2 -23039.999} C_VEL
LIN {X 0,Y 171.785,Z 324.063,A -85,B 0,C 180,E1 -23044.693,E2 -23044.693} C_VEL
LIN {X 0,Y 171.847,Z 324.071,A -85,B 0,C 180,E1 -23049.415,E2 -23049.415} C_VEL
LIN {X 0,Y 171.561,Z 324.109,A -85,B 0,C 180,E1 -23054.228,E2 -23054.228} C_VEL
LIN {X 0,Y 171.484,Z 324.123,A -85,B 0,C 180,E1 -23059.499,E2 -23059.499} C_VEL
LIN {X 0,Y 171.447,Z 324.13,A -85,B 0,C 180,E1 -23065.597,E2 -23065.597} C_VEL
LIN {X 0,Y 171.421,Z 324.131,A -85,B 0,C 180,E1 -23070.571,E2 -23070.571} C_VEL
LIN {X 0,Y 171.395,Z 324.138,A -85,B 0,C 180,E1 -23075.034,E2 -23075.034} C_VEL
LIN {X 0,Y 171.345,Z 324.143,A -85,B 0,C 180,E1 -23078.8,E2 -23078.8} C_VEL
LIN {X 0,Y 171.358,Z 324.28,A -85,B 0,C 180,E1 -23084.205,E2 -23084.205} C_VEL
LIN {X 0,Y 172.359,Z 327.987,A -85,B 0,C 180,E1 -23086.499,E2 -23086.499} C_VEL
LIN {X 0,Y 174.691,Z 332.386,A -85,B 0,C 180,E1 -23087.347,E2 -23087.347} C_VEL
LIN {X 0,Y 179.956,Z 342.823,A -85,B 0,C 180,E1 -23089.171,E2 -23089.171} C_VEL
LIN {X 0,Y 185.392,Z 355.13,A -85,B 0,C 180,E1 -23090.977,E2 -23090.977} C_VEL
LIN {X 0,Y 189.652,Z 366.726,A -85,B 0,C 180,E1 -23092.382,E2 -23092.382} C_VEL
LIN {X 0,Y 191.883,Z 391.697,A -85,B 0,C 180,E1 -23093.907,E2 -23093.907} C_VEL
LIN {X 0,Y 189.749,Z 438.262,A -85,B 0,C 180,E1 -23095.605,E2 -23095.605} C_VEL
LIN {X 0,Y 188.267,Z 452.18,A -85,B 0,C 180,E1 -23096.509,E2 -23096.509} C_VEL
LIN {X 0,Y 186.2,Z 465.099,A -85,B 0,C 180,E1 -23097.781,E2 -23097.781} C_VEL
LIN {X 0,Y 183.741,Z 477.33,A -85,B 0,C 180,E1 -23099.473,E2 -23099.473} C_VEL
LIN {X 0,Y 181.949,Z 482.428,A -85,B 0,C 180,E1 -23100.242,E2 -23100.242} C_VEL
LIN {X 0,Y 177.263,Z 490.314,A -85,B 0,C 180,E1 -23101.449,E2 -23101.449} C_VEL
LIN {X 0,Y 172.548,Z 497.777,A -85,B 0,C 180,E1 -23102.912,E2 -23102.912} C_VEL
LIN {X 0,Y 170.715,Z 502.145,A -85,B 0,C 180,E1 -23104.096,E2 -23104.096} C_VEL
LIN {X 0,Y 168.55,Z 509.529,A -85,B 0,C 180,E1 -23106.538,E2 -23106.538} C_VEL
LIN {X 0,Y 166.444,Z 517.059,A -85,B 0,C 180,E1 -23109.612,E2 -23109.612} C_VEL
LIN {X 0,Y 164.454,Z 524.107,A -85,B 0,C 180,E1 -23113.232,E2 -23113.232} C_VEL
LIN {X 0,Y 162.855,Z 530.559,A -85,B 0,C 180,E1 -23117.537,E2 -23117.537} C_VEL
LIN {X 0,Y 162.19,Z 534.791,A -85,B 0,C 180,E1 -23121.275,E2 -23121.275} C_VEL
LIN {X 0,Y 161.987,Z 538.764,A -85,B 0,C 180,E1 -23126.268,E2 -23126.268} C_VEL
LIN {X 0,Y 162.177,Z 540.595,A -85,B 0,C 180,E1 -23129.998,E2 -23129.998} C_VEL
LIN {X 0,Y 161.912,Z 541.394,A -85,B 0,C 180,E1 -23133.299,E2 -23133.299} C_VEL
LIN {X 0,Y 162.003,Z 541.407,A -85,B 0,C 180,E1 -23137.476,E2 -23137.476} C_VEL
LIN {X 0,Y 162.356,Z 540.889,A -85,B 0,C 180,E1 -23139.969,E2 -23139.969} C_VEL
LIN {X 0,Y 163.82,Z 538.635,A -85,B 0,C 180,E1 -23144.915,E2 -23144.915} C_VEL
LIN {X 0,Y 165.768,Z 535.88,A -85,B 0,C 180,E1 -23148.539,E2 -23148.539} C_VEL
LIN {X 0,Y 168.355,Z 532.128,A -85,B 0,C 180,E1 -23152.066,E2 -23152.066} C_VEL
LIN {X 0,Y 172.257,Z 526.168,A -85,B 0,C 180,E1 -23156.158,E2 -23156.158} C_VEL
LIN {X 0,Y 176.662,Z 518.863,A -85,B 0,C 180,E1 -23159.818,E2 -23159.818} C_VEL
LIN {X 0,Y 181.312,Z 510.742,A -85,B 0,C 180,E1 -23162.864,E2 -23162.864} C_VEL
LIN {X 0,Y 185.557,Z 502.475,A -85,B 0,C 180,E1 -23165.28,E2 -23165.28} C_VEL
LIN {X 0,Y 189.74,Z 493.482,A -85,B 0,C 180,E1 -23167.338,E2 -23167.338} C_VEL
LIN {X 0,Y 193.152,Z 485.072,A -85,B 0,C 180,E1 -23168.876,E2 -23168.876} C_VEL
LIN {X 0,Y 197.267,Z 473.31,A -85,B 0,C 180,E1 -23170.554,E2 -23170.554} C_VEL
LIN {X 0,Y 200.507,Z 461.846,A -85,B 0,C 180,E1 -23171.755,E2 -23171.755} C_VEL
LIN {X 0,Y 203.369,Z 448.301,A -85,B 0,C 180,E1 -23172.773,E2 -23172.773} C_VEL
LIN {X 0,Y 205.031,Z 435.892,A -85,B 0,C 180,E1 -23173.405,E2 -23173.405} C_VEL
LIN {X 0,Y 207.494,Z 400.322,A -85,B 0,C 180,E1 -23174.515,E2 -23174.515} C_VEL
LIN {X 0,Y 206.962,Z 396.481,A -85,B 0,C 180,E1 -23174.878,E2 -23174.878} C_VEL
LIN {X 0,Y 202.248,Z 384.699,A -85,B 0,C 180,E1 -23177.062,E2 -23177.062} C_VEL
LIN {X 0,Y 197.181,Z 373.916,A -85,B 0,C 180,E1 -23179.546,E2 -23179.546} C_VEL
LIN {X 0,Y 192.114,Z 364.483,A -85,B 0,C 180,E1 -23182.244,E2 -23182.244} C_VEL
LIN {X 0,Y 188.512,Z 358.321,A -85,B 0,C 180,E1 -23184.34,E2 -23184.34} C_VEL
LIN {X 0,Y 186.344,Z 354.696,A -85,B 0,C 180,E1 -23185.704,E2 -23185.704} C_VEL
LIN {X 0,Y 183.192,Z 349.622,A -85,B 0,C 180,E1 -23187.839,E2 -23187.839} C_VEL
LIN {X 0,Y 179.185,Z 343.668,A -85,B 0,C 180,E1 -23190.87,E2 -23190.87} C_VEL
LIN {X 0,Y 174.611,Z 337.257,A -85,B 0,C 180,E1 -23194.981,E2 -23194.981} C_VEL
LIN {X 0,Y 173.205,Z 335.95,A -85,B 0,C 180,E1 -23196.379,E2 -23196.379} C_VEL
LIN {X 0,Y 170.978,Z 333.658,A -85,B 0,C 180,E1 -23198.921,E2 -23198.921} C_VEL
LIN {X 0,Y 169.819,Z 330.989,A -85,B 0,C 180,E1 -23200.666,E2 -23200.666} C_VEL
LIN {X 0,Y 166.594,Z 329.15,A -85,B 0,C 180,E1 -23205.9,E2 -23205.9} C_VEL
LIN {X 0,Y 164.855,Z 324.94,A -85,B 0,C 180,E1 -23212.807,E2 -23212.807} C_VEL
LIN {X 0,Y 165.293,Z 324.884,A -85,B 0,C 180,E1 -23220.001,E2 -23220.001} C_VEL
LIN {X 0,Y 165.196,Z 325.081,A -85,B 0,C 180,E1 -23220.839,E2 -23220.839} C_VEL
LIN {X 0,Y 165.894,Z 327.887,A -85,B 0,C 180,E1 -23223.948,E2 -23223.948} C_VEL
LIN {X 0,Y 168.788,Z 330.446,A -85,B 0,C 180,E1 -23229.588,E2 -23229.588} C_VEL
LIN {X 0,Y 170.132,Z 331.179,A -85,B 0,C 180,E1 -23231.43,E2 -23231.43} C_VEL
LIN {X 0,Y 171.453,Z 334.077,A -85,B 0,C 180,E1 -23233.332,E2 -23233.332} C_VEL
LIN {X 0,Y 173.764,Z 336.235,A -85,B 0,C 180,E1 -23235.844,E2 -23235.844} C_VEL
LIN {X 0,Y 174.911,Z 337.119,A -85,B 0,C 180,E1 -23236.937,E2 -23236.937} C_VEL
LIN {X 0,Y 176.721,Z 340.17,A -85,B 0,C 180,E1 -23238.702,E2 -23238.702} C_VEL
LIN {X 0,Y 179.318,Z 342.657,A -85,B 0,C 180,E1 -23240.806,E2 -23240.806} C_VEL
LIN {X 0,Y 181.923,Z 346.293,A -85,B 0,C 180,E1 -23242.805,E2 -23242.805} C_VEL
LIN {X 0,Y 183.28,Z 347.817,A -85,B 0,C 180,E1 -23243.744,E2 -23243.744} C_VEL
LIN {X 0,Y 187.03,Z 352.925,A -85,B 0,C 180,E1 -23246.202,E2 -23246.202} C_VEL
LIN {X 0,Y 190.742,Z 358.194,A -85,B 0,C 180,E1 -23248.395,E2 -23248.395} C_VEL
LIN {X 0,Y 195.016,Z 364.358,A -85,B 0,C 180,E1 -23250.676,E2 -23250.676} C_VEL
LIN {X 0,Y 201.21,Z 374.4,A -85,B 0,C 180,E1 -23253.677,E2 -23253.677} C_VEL
LIN {X 0,Y 207.621,Z 386.168,A -85,B 0,C 180,E1 -23256.478,E2 -23256.478} C_VEL
LIN {X 0,Y 208.287,Z 387.513,A -85,B 0,C 180,E1 -23256.756,E2 -23256.756} C_VEL
LIN {X 0,Y 205.678,Z 424.022,A -85,B 0,C 180,E1 -23257.899,E2 -23257.899} C_VEL
LIN {X 0,Y 203.921,Z 437.297,A -85,B 0,C 180,E1 -23258.66,E2 -23258.66} C_VEL
LIN {X 0,Y 201.506,Z 449.637,A -85,B 0,C 180,E1 -23259.711,E2 -23259.711} C_VEL
LIN {X 0,Y 198.068,Z 461.729,A -85,B 0,C 180,E1 -23261.063,E2 -23261.063} C_VEL
LIN {X 0,Y 194.152,Z 473.334,A -85,B 0,C 180,E1 -23262.862,E2 -23262.862} C_VEL
LIN {X 0,Y 190.419,Z 483.079,A -85,B 0,C 180,E1 -23264.866,E2 -23264.866} C_VEL
LIN {X 0,Y 186.178,Z 492.197,A -85,B 0,C 180,E1 -23267.199,E2 -23267.199} C_VEL
LIN {X 0,Y 181.343,Z 501.321,A -85,B 0,C 180,E1 -23270.25,E2 -23270.25} C_VEL
LIN {X 0,Y 177.03,Z 508.632,A -85,B 0,C 180,E1 -23273.454,E2 -23273.454} C_VEL
LIN {X 0,Y 173.15,Z 514.431,A -85,B 0,C 180,E1 -23276.775,E2 -23276.775} C_VEL
LIN {X 0,Y 169.77,Z 519.107,A -85,B 0,C 180,E1 -23280.384,E2 -23280.384} C_VEL
LIN {X 0,Y 168.043,Z 521.32,A -85,B 0,C 180,E1 -23282.612,E2 -23282.612} C_VEL
LIN {X 0,Y 166.402,Z 523.246,A -85,B 0,C 180,E1 -23285.019,E2 -23285.019} C_VEL
LIN {X 0,Y 165.085,Z 524.737,A -85,B 0,C 180,E1 -23287.473,E2 -23287.473} C_VEL
LIN {X 0,Y 163.152,Z 526.394,A -85,B 0,C 180,E1 -23292.452,E2 -23292.452} C_VEL
LIN {X 0,Y 162.511,Z 526.636,A -85,B 0,C 180,E1 -23294.963,E2 -23294.963} C_VEL
LIN {X 0,Y 162.065,Z 526.474,A -85,B 0,C 180,E1 -23297.479,E2 -23297.479} C_VEL
LIN {X 0,Y 161.955,Z 524.891,A -85,B 0,C 180,E1 -23302.521,E2 -23302.521} C_VEL
LIN {X 0,Y 162.226,Z 523.438,A -85,B 0,C 180,E1 -23305.159,E2 -23305.159} C_VEL
LIN {X 0,Y 162.652,Z 520.642,A -85,B 0,C 180,E1 -23308.764,E2 -23308.764} C_VEL
LIN {X 0,Y 163.545,Z 516.753,A -85,B 0,C 180,E1 -23312.464,E2 -23312.464} C_VEL
LIN {X 0,Y 164.932,Z 511.74,A -85,B 0,C 180,E1 -23316.117,E2 -23316.117} C_VEL
LIN {X 0,Y 166.787,Z 505.45,A -85,B 0,C 180,E1 -23319.705,E2 -23319.705} C_VEL
LIN {X 0,Y 169.207,Z 497.572,A -85,B 0,C 180,E1 -23323.207,E2 -23323.207} C_VEL
LIN {X 0,Y 171.635,Z 489.547,A -85,B 0,C 180,E1 -23326.047,E2 -23326.047} C_VEL
LIN {X 0,Y 174.473,Z 479.752,A -85,B 0,C 180,E1 -23328.801,E2 -23328.801} C_VEL
LIN {X 0,Y 177.271,Z 468.793,A -85,B 0,C 180,E1 -23331.21,E2 -23331.21} C_VEL
LIN {X 0,Y 179.555,Z 458.075,A -85,B 0,C 180,E1 -23333.044,E2 -23333.044} C_VEL
LIN {X 0,Y 181.508,Z 446.324,A -85,B 0,C 180,E1 -23334.599,E2 -23334.599} C_VEL
LIN {X 0,Y 183.196,Z 433.724,A -85,B 0,C 180,E1 -23335.789,E2 -23335.789} C_VEL
LIN {X 0,Y 184.269,Z 420.565,A -85,B 0,C 180,E1 -23336.593,E2 -23336.593} C_VEL
LIN {X 0,Y 186.956,Z 366.827,A -85,B 0,C 180,E1 -23338.524,E2 -23338.524} C_VEL
LIN {X 0,Y 180.446,Z 352.952,A -85,B 0,C 180,E1 -23340.59,E2 -23340.59} C_VEL
LIN {X 0,Y 175.237,Z 343.322,A -85,B 0,C 180,E1 -23342.32,E2 -23342.32} C_VEL
LIN {X 0,Y 168.864,Z 332.915,A -85,B 0,C 180,E1 -23344.567,E2 -23344.567} C_VEL
LIN {X 0,Y 166.611,Z 329.37,A -85,B 0,C 180,E1 -23345.413,E2 -23345.413} C_VEL
LIN {X 0,Y 164.852,Z 327.008,A -85,B 0,C 180,E1 -23346.074,E2 -23346.074} C_VEL
LIN {X 0,Y 164.297,Z 325.019,A -85,B 0,C 180,E1 -23346.399,E2 -23346.399} C_VEL
LIN {X 0,Y 164.29,Z 325.009,A -85,B 0,C 180,E1 -23349.918,E2 -23349.918} C_VEL
LIN {X 0,Y 164.285,Z 325.017,A -85,B 0,C 180,E1 -23353.342,E2 -23353.342} C_VEL
LIN {X 0,Y 164.264,Z 325.004,A -85,B 0,C 180,E1 -23356.798,E2 -23356.798} C_VEL
LIN {X 0,Y 164.294,Z 325.016,A -85,B 0,C 180,E1 -23360.355,E2 -23360.355} C_VEL
LIN {X 0,Y 164.33,Z 324.994,A -85,B 0,C 180,E1 -23364.352,E2 -23364.352} C_VEL
LIN {X 0,Y 164.375,Z 325.008,A -85,B 0,C 180,E1 -23369.131,E2 -23369.131} C_VEL
LIN {X 0,Y 164.399,Z 324.977,A -85,B 0,C 180,E1 -23374.69,E2 -23374.69} C_VEL
LIN {X 0,Y 164.49,Z 324.995,A -85,B 0,C 180,E1 -23380.052,E2 -23380.052} C_VEL
LIN {X 0,Y 164.502,Z 324.962,A -85,B 0,C 180,E1 -23385.146,E2 -23385.146} C_VEL
LIN {X 0,Y 164.77,Z 324.96,A -85,B 0,C 180,E1 -23390.176,E2 -23390.176} C_VEL
LIN {X 0,Y 164.826,Z 324.941,A -85,B 0,C 180,E1 -23392.65,E2 -23392.65} C_VEL
LIN {X 0,Y 165.278,Z 324.894,A -85,B 0,C 180,E1 -23399.999,E2 -23399.999} C_VEL
LIN {X 0,Y 164.823,Z 324.925,A -85,B 0,C 180,E1 -23407.349,E2 -23407.349} C_VEL
LIN {X 0,Y 164.706,Z 324.969,A -85,B 0,C 180,E1 -23411.058,E2 -23411.058} C_VEL
LIN {X 0,Y 164.442,Z 324.999,A -85,B 0,C 180,E1 -23417.407,E2 -23417.407} C_VEL
LIN {X 0,Y 164.355,Z 325.009,A -85,B 0,C 180,E1 -23422.634,E2 -23422.634} C_VEL
LIN {X 0,Y 164.373,Z 325.011,A -85,B 0,C 180,E1 -23426.115,E2 -23426.115} C_VEL
LIN {X 0,Y 164.36,Z 325.01,A -85,B 0,C 180,E1 -23431.216,E2 -23431.216} C_VEL
LIN {X 0,Y 164.282,Z 325.024,A -85,B 0,C 180,E1 -23436.792,E2 -23436.792} C_VEL
LIN {X 0,Y 164.276,Z 325.023,A -85,B 0,C 180,E1 -23441.537,E2 -23441.537} C_VEL
LIN {X 0,Y 164.314,Z 325.137,A -85,B 0,C 180,E1 -23442.765,E2 -23442.765} C_VEL
LIN {X 0,Y 164.946,Z 327.486,A -85,B 0,C 180,E1 -23444.347,E2 -23444.347} C_VEL
LIN {X 0,Y 167.537,Z 332.254,A -85,B 0,C 180,E1 -23445.383,E2 -23445.383} C_VEL
LIN {X 0,Y 173.121,Z 342.89,A -85,B 0,C 180,E1 -23447.482,E2 -23447.482} C_VEL
LIN {X 0,Y 178.137,Z 353.839,A -85,B 0,C 180,E1 -23449.281,E2 -23449.281} C_VEL
LIN {X 0,Y 183.417,Z 367.705,A -85,B 0,C 180,E1 -23451.138,E2 -23451.138} C_VEL
LIN {X 0,Y 183.994,Z 370.602,A -85,B 0,C 180,E1 -23451.397,E2 -23451.397} C_VEL
LIN {X 0,Y 185.858,Z 392.151,A -85,B 0,C 180,E1 -23452.768,E2 -23452.768} C_VEL
LIN {X 0,Y 183.676,Z 437.947,A -85,B 0,C 180,E1 -23454.486,E2 -23454.486} C_VEL
LIN {X 0,Y 182.166,Z 451.682,A -85,B 0,C 180,E1 -23455.398,E2 -23455.398} C_VEL
LIN {X 0,Y 179.982,Z 464.652,A -85,B 0,C 180,E1 -23456.692,E2 -23456.692} C_VEL
LIN {X 0,Y 177.545,Z 476.484,A -85,B 0,C 180,E1 -23458.364,E2 -23458.364} C_VEL
LIN {X 0,Y 174.661,Z 487.869,A -85,B 0,C 180,E1 -23460.466,E2 -23460.466} C_VEL
LIN {X 0,Y 171.902,Z 498.142,A -85,B 0,C 180,E1 -23462.944,E2 -23462.944} C_VEL
LIN {X 0,Y 170.715,Z 502.145,A -85,B 0,C 180,E1 -23464.096,E2 -23464.096} C_VEL
LIN {X 0,Y 168.934,Z 506.363,A -85,B 0,C 180,E1 -23465.367,E2 -23465.367} C_VEL
LIN {X 0,Y 162.381,Z 515.089,A -85,B 0,C 180,E1 -23468.345,E2 -23468.345} C_VEL
LIN {X 0,Y 159.103,Z 519.62,A -85,B 0,C 180,E1 -23470.354,E2 -23470.354} C_VEL
LIN {X 0,Y 158.132,Z 521.761,A -85,B 0,C 180,E1 -23471.495,E2 -23471.495} C_VEL
LIN {X 0,Y 156.267,Z 528.333,A -85,B 0,C 180,E1 -23475.677,E2 -23475.677} C_VEL
LIN {X 0,Y 155.333,Z 533.008,A -85,B 0,C 180,E1 -23479.572,E2 -23479.572} C_VEL
LIN {X 0,Y 154.907,Z 536.55,A -85,B 0,C 180,E1 -23483.486,E2 -23483.486} C_VEL
LIN {X 0,Y 154.932,Z 539.062,A -85,B 0,C 180,E1 -23487.398,E2 -23487.398} C_VEL
LIN {X 0,Y 155.096,Z 540.209,A -85,B 0,C 180,E1 -23489.998,E2 -23489.998} C_VEL
LIN {X 0,Y 154.854,Z 540.987,A -85,B 0,C 180,E1 -23493.185,E2 -23493.185} C_VEL
LIN {X 0,Y 154.947,Z 541.086,A -85,B 0,C 180,E1 -23497.819,E2 -23497.819} C_VEL
LIN {X 0,Y 155.331,Z 540.607,A -85,B 0,C 180,E1 -23500.425,E2 -23500.425} C_VEL
LIN {X 0,Y 156.929,Z 538.403,A -85,B 0,C 180,E1 -23505.586,E2 -23505.586} C_VEL
LIN {X 0,Y 159.026,Z 535.696,A -85,B 0,C 180,E1 -23509.355,E2 -23509.355} C_VEL
LIN {X 0,Y 161.783,Z 531.995,A -85,B 0,C 180,E1 -23513.013,E2 -23513.013} C_VEL
LIN {X 0,Y 165.536,Z 526.592,A -85,B 0,C 180,E1 -23516.929,E2 -23516.929} C_VEL
LIN {X 0,Y 169.798,Z 520.061,A -85,B 0,C 180,E1 -23520.464,E2 -23520.464} C_VEL
LIN {X 0,Y 174.526,Z 512.319,A -85,B 0,C 180,E1 -23523.62,E2 -23523.62} C_VEL
LIN {X 0,Y 179.823,Z 502.649,A -85,B 0,C 180,E1 -23526.583,E2 -23526.583} C_VEL
LIN {X 0,Y 184.166,Z 493.756,A -85,B 0,C 180,E1 -23528.672,E2 -23528.672} C_VEL
LIN {X 0,Y 187.692,Z 485.473,A -85,B 0,C 180,E1 -23530.232,E2 -23530.232} C_VEL
LIN {X 0,Y 191.944,Z 473.911,A -85,B 0,C 180,E1 -23531.928,E2 -23531.928} C_VEL
LIN {X 0,Y 195.3,Z 462.785,A -85,B 0,C 180,E1 -23533.134,E2 -23533.134} C_VEL
LIN {X 0,Y 198.21,Z 449.958,A -85,B 0,C 180,E1 -23534.137,E2 -23534.137} C_VEL
LIN {X 0,Y 200.196,Z 436.468,A -85,B 0,C 180,E1 -23534.863,E2 -23534.863} C_VEL
LIN {X 0,Y 202.761,Z 401.516,A -85,B 0,C 180,E1 -23535.971,E2 -23535.971} C_VEL
LIN {X 0,Y 202.34,Z 399.285,A -85,B 0,C 180,E1 -23536.232,E2 -23536.232} C_VEL
LIN {X 0,Y 197.411,Z 386.922,A -85,B 0,C 180,E1 -23538.685,E2 -23538.685} C_VEL
LIN {X 0,Y 192.457,Z 376.361,A -85,B 0,C 180,E1 -23541.322,E2 -23541.322} C_VEL
LIN {X 0,Y 188.769,Z 369.424,A -85,B 0,C 180,E1 -23543.439,E2 -23543.439} C_VEL
LIN {X 0,Y 184.343,Z 361.429,A -85,B 0,C 180,E1 -23546.258,E2 -23546.258} C_VEL
LIN {X 0,Y 180.484,Z 355.176,A -85,B 0,C 180,E1 -23549.004,E2 -23549.004} C_VEL
LIN {X 0,Y 177.029,Z 349.832,A -85,B 0,C 180,E1 -23551.792,E2 -23551.792} C_VEL
LIN {X 0,Y 172.838,Z 343.697,A -85,B 0,C 180,E1 -23555.792,E2 -23555.792} C_VEL
LIN {X 0,Y 169.548,Z 340.366,A -85,B 0,C 180,E1 -23559.549,E2 -23559.549} C_VEL
LIN {X 0,Y 168.485,Z 337.95,A -85,B 0,C 180,E1 -23561.22,E2 -23561.22} C_VEL
LIN {X 0,Y 165.324,Z 335.813,A -85,B 0,C 180,E1 -23566.783,E2 -23566.783} C_VEL
LIN {X 0,Y 163.882,Z 331.966,A -85,B 0,C 180,E1 -23573.228,E2 -23573.228} C_VEL
LIN {X 0,Y 164.207,Z 332.044,A -85,B 0,C 180,E1 -23580.307,E2 -23580.307} C_VEL
LIN {X 0,Y 164.908,Z 334.883,A -85,B 0,C 180,E1 -23583.666,E2 -23583.666} C_VEL
LIN {X 0,Y 167.529,Z 337.323,A -85,B 0,C 180,E1 -23589.052,E2 -23589.052} C_VEL
LIN {X 0,Y 168.699,Z 338.032,A -85,B 0,C 180,E1 -23590.752,E2 -23590.752} C_VEL
LIN {X 0,Y 170.207,Z 341.089,A -85,B 0,C 180,E1 -23592.975,E2 -23592.975} C_VEL
LIN {X 0,Y 173.198,Z 343.783,A -85,B 0,C 180,E1 -23596.219,E2 -23596.219} C_VEL
LIN {X 0,Y 175.236,Z 347.008,A -85,B 0,C 180,E1 -23598.261,E2 -23598.261} C_VEL
LIN {X 0,Y 177.399,Z 349.242,A -85,B 0,C 180,E1 -23600.094,E2 -23600.094} C_VEL
LIN {X 0,Y 180.157,Z 352.971,A -85,B 0,C 180,E1 -23602.281,E2 -23602.281} C_VEL
LIN {X 0,Y 184.481,Z 358.872,A -85,B 0,C 180,E1 -23605.299,E2 -23605.299} C_VEL
LIN {X 0,Y 189.827,Z 366.61,A -85,B 0,C 180,E1 -23608.545,E2 -23608.545} C_VEL
LIN {X 0,Y 195.71,Z 376.028,A -85,B 0,C 180,E1 -23611.682,E2 -23611.682} C_VEL
LIN {X 0,Y 201.257,Z 386.024,A -85,B 0,C 180,E1 -23614.347,E2 -23614.347} C_VEL
LIN {X 0,Y 203.478,Z 390.371,A -85,B 0,C 180,E1 -23615.35,E2 -23615.35} C_VEL
LIN {X 0,Y 200.898,Z 424.611,A -85,B 0,C 180,E1 -23616.43,E2 -23616.43} C_VEL
LIN {X 0,Y 199.065,Z 437.84,A -85,B 0,C 180,E1 -23617.199,E2 -23617.199} C_VEL
LIN {X 0,Y 196.457,Z 450.548,A -85,B 0,C 180,E1 -23618.301,E2 -23618.301} C_VEL
LIN {X 0,Y 192.88,Z 462.553,A -85,B 0,C 180,E1 -23619.672,E2 -23619.672} C_VEL
LIN {X 0,Y 188.811,Z 474.066,A -85,B 0,C 180,E1 -23621.49,E2 -23621.49} C_VEL
LIN {X 0,Y 184.61,Z 484.386,A -85,B 0,C 180,E1 -23623.673,E2 -23623.673} C_VEL
LIN {X 0,Y 180.042,Z 493.604,A -85,B 0,C 180,E1 -23626.144,E2 -23626.144} C_VEL
LIN {X 0,Y 175.012,Z 502.545,A -85,B 0,C 180,E1 -23629.267,E2 -23629.267} C_VEL
LIN {X 0,Y 170.529,Z 509.66,A -85,B 0,C 180,E1 -23632.565,E2 -23632.565} C_VEL
LIN {X 0,Y 165.898,Z 516.103,A -85,B 0,C 180,E1 -23636.585,E2 -23636.585} C_VEL
LIN {X 0,Y 163.207,Z 519.561,A -85,B 0,C 180,E1 -23639.458,E2 -23639.458} C_VEL
LIN {X 0,Y 159.849,Z 523.423,A -85,B 0,C 180,E1 -23643.919,E2 -23643.919} C_VEL
LIN {X 0,Y 158.393,Z 524.955,A -85,B 0,C 180,E1 -23646.465,E2 -23646.465} C_VEL
LIN {X 0,Y 156.713,Z 526.418,A -85,B 0,C 180,E1 -23650.354,E2 -23650.354} C_VEL
LIN {X 0,Y 155.558,Z 526.957,A -85,B 0,C 180,E1 -23654.273,E2 -23654.273} C_VEL
LIN {X 0,Y 155.039,Z 526.84,A -85,B 0,C 180,E1 -23656.902,E2 -23656.902} C_VEL
LIN {X 0,Y 154.82,Z 526.283,A -85,B 0,C 180,E1 -23659.54,E2 -23659.54} C_VEL
LIN {X 0,Y 155.101,Z 523.975,A -85,B 0,C 180,E1 -23664.802,E2 -23664.802} C_VEL
LIN {X 0,Y 155.56,Z 521.159,A -85,B 0,C 180,E1 -23668.707,E2 -23668.707} C_VEL
LIN {X 0,Y 156.436,Z 517.335,A -85,B 0,C 180,E1 -23672.577,E2 -23672.577} C_VEL
LIN {X 0,Y 157.88,Z 512.389,A -85,B 0,C 180,E1 -23676.391,E2 -23676.391} C_VEL
LIN {X 0,Y 159.819,Z 506.182,A -85,B 0,C 180,E1 -23680.133,E2 -23680.133} C_VEL
LIN {X 0,Y 162.338,Z 498.422,A -85,B 0,C 180,E1 -23683.776,E2 -23683.776} C_VEL
LIN {X 0,Y 165.389,Z 488.73,A -85,B 0,C 180,E1 -23687.306,E2 -23687.306} C_VEL
LIN {X 0,Y 168.406,Z 478.675,A -85,B 0,C 180,E1 -23690.14,E2 -23690.14} C_VEL
LIN {X 0,Y 171.391,Z 467.286,A -85,B 0,C 180,E1 -23692.61,E2 -23692.61} C_VEL
LIN {X 0,Y 173.779,Z 456.138,A -85,B 0,C 180,E1 -23694.491,E2 -23694.491} C_VEL
LIN {X 0,Y 175.701,Z 444.862,A -85,B 0,C 180,E1 -23695.946,E2 -23695.946} C_VEL
LIN {X 0,Y 177.384,Z 431.746,A -85,B 0,C 180,E1 -23697.134,E2 -23697.134} C_VEL
LIN {X 0,Y 178.388,Z 418.724,A -85,B 0,C 180,E1 -23697.885,E2 -23697.885} C_VEL
LIN {X 0,Y 180.995,Z 368.816,A -85,B 0,C 180,E1 -23699.704,E2 -23699.704} C_VEL
LIN {X 0,Y 174.124,Z 354.183,A -85,B 0,C 180,E1 -23702.046,E2 -23702.046} C_VEL
LIN {X 0,Y 166.638,Z 341.127,A -85,B 0,C 180,E1 -23704.751,E2 -23704.751} C_VEL
LIN {X 0,Y 162.252,Z 334.336,A -85,B 0,C 180,E1 -23706.457,E2 -23706.457} C_VEL
LIN {X 0,Y 159.723,Z 330.481,A -85,B 0,C 180,E1 -23707.501,E2 -23707.501} C_VEL
LIN {X 0,Y 157.888,Z 328.168,A -85,B 0,C 180,E1 -23708.262,E2 -23708.262} C_VEL
LIN {X 0,Y 157.206,Z 325.902,A -85,B 0,C 180,E1 -23708.65,E2 -23708.65} C_VEL
LIN {X 0,Y 157.184,Z 325.903,A -85,B 0,C 180,E1 -23714.323,E2 -23714.323} C_VEL
LIN {X 0,Y 157.198,Z 325.892,A -85,B 0,C 180,E1 -23719.47,E2 -23719.47} C_VEL
LIN {X 0,Y 157.279,Z 325.87,A -85,B 0,C 180,E1 -23724.485,E2 -23724.485} C_VEL
LIN {X 0,Y 157.288,Z 325.884,A -85,B 0,C 180,E1 -23728.102,E2 -23728.102} C_VEL
LIN {X 0,Y 157.314,Z 325.863,A -85,B 0,C 180,E1 -23733.464,E2 -23733.464} C_VEL
LIN {X 0,Y 157.397,Z 325.88,A -85,B 0,C 180,E1 -23739.67,E2 -23739.67} C_VEL
LIN {X 0,Y 157.44,Z 325.84,A -85,B 0,C 180,E1 -23744.464,E2 -23744.464} C_VEL
LIN {X 0,Y 157.693,Z 325.841,A -85,B 0,C 180,E1 -23749.73,E2 -23749.73} C_VEL
LIN {X 0,Y 157.764,Z 325.822,A -85,B 0,C 180,E1 -23752.319,E2 -23752.319} C_VEL
LIN {X 0,Y 158.241,Z 325.771,A -85,B 0,C 180,E1 -23759.999,E2 -23759.999} C_VEL
LIN {X 0,Y 157.762,Z 325.805,A -85,B 0,C 180,E1 -23767.68,E2 -23767.68} C_VEL
LIN {X 0,Y 157.637,Z 325.849,A -85,B 0,C 180,E1 -23771.226,E2 -23771.226} C_VEL
LIN {X 0,Y 157.421,Z 325.876,A -85,B 0,C 180,E1 -23775.537,E2 -23775.537} C_VEL
LIN {X 0,Y 157.315,Z 325.891,A -85,B 0,C 180,E1 -23780.94,E2 -23780.94} C_VEL
LIN {X 0,Y 157.313,Z 325.887,A -85,B 0,C 180,E1 -23786.68,E2 -23786.68} C_VEL
LIN {X 0,Y 157.271,Z 325.897,A -85,B 0,C 180,E1 -23792.428,E2 -23792.428} C_VEL
LIN {X 0,Y 157.261,Z 325.899,A -85,B 0,C 180,E1 -23796.443,E2 -23796.443} C_VEL
LIN {X 0,Y 157.256,Z 326.055,A -85,B 0,C 180,E1 -23801.203,E2 -23801.203} C_VEL
LIN {X 0,Y 157.497,Z 327.083,A -85,B 0,C 180,E1 -23801.904,E2 -23801.904} C_VEL
LIN {X 0,Y 159.811,Z 331.28,A -85,B 0,C 180,E1 -23802.943,E2 -23802.943} C_VEL
LIN {X 0,Y 161.058,Z 333.319,A -85,B 0,C 180,E1 -23803.47,E2 -23803.47} C_VEL
LIN {X 0,Y 166.852,Z 344.086,A -85,B 0,C 180,E1 -23805.838,E2 -23805.838} C_VEL
LIN {X 0,Y 172.534,Z 356.232,A -85,B 0,C 180,E1 -23808.021,E2 -23808.021} C_VEL
LIN {X 0,Y 177.993,Z 370.854,A -85,B 0,C 180,E1 -23810.081,E2 -23810.081} C_VEL
LIN {X 0,Y 179.283,Z 384.425,A -85,B 0,C 180,E1 -23811.028,E2 -23811.028} C_VEL
LIN {X 0,Y 179.926,Z 394.462,A -85,B 0,C 180,E1 -23811.646,E2 -23811.646} C_VEL
LIN {X 0,Y 177.663,Z 437.321,A -85,B 0,C 180,E1 -23813.265,E2 -23813.265} C_VEL
LIN {X 0,Y 176.118,Z 451.178,A -85,B 0,C 180,E1 -23814.205,E2 -23814.205} C_VEL
LIN {X 0,Y 174.084,Z 463.152,A -85,B 0,C 180,E1 -23815.407,E2 -23815.407} C_VEL
LIN {X 0,Y 171.463,Z 475.258,A -85,B 0,C 180,E1 -23817.104,E2 -23817.104} C_VEL
LIN {X 0,Y 168.526,Z 486.822,A -85,B 0,C 180,E1 -23819.277,E2 -23819.277} C_VEL
LIN {X 0,Y 165.507,Z 497.234,A -85,B 0,C 180,E1 -23821.808,E2 -23821.808} C_VEL
LIN {X 0,Y 162.984,Z 505.755,A -85,B 0,C 180,E1 -23824.454,E2 -23824.454} C_VEL
LIN {X 0,Y 160.593,Z 513.605,A -85,B 0,C 180,E1 -23827.483,E2 -23827.483} C_VEL
LIN {X 0,Y 158.132,Z 521.761,A -85,B 0,C 180,E1 -23831.495,E2 -23831.495} C_VEL
LIN {X 0,Y 156.582,Z 524.81,A -85,B 0,C 180,E1 -23833.255,E2 -23833.255} C_VEL
LIN {X 0,Y 152.578,Z 529.155,A -85,B 0,C 180,E1 -23836.211,E2 -23836.211} C_VEL
LIN {X 0,Y 148.933,Z 532.856,A -85,B 0,C 180,E1 -23839.437,E2 -23839.437} C_VEL
LIN {X 0,Y 147.984,Z 534.776,A -85,B 0,C 180,E1 -23841.558,E2 -23841.558} C_VEL
LIN {X 0,Y 147.838,Z 538.303,A -85,B 0,C 180,E1 -23846.66,E2 -23846.66} C_VEL
LIN {X 0,Y 148.015,Z 539.817,A -85,B 0,C 180,E1 -23849.998,E2 -23849.998} C_VEL
LIN {X 0,Y 147.79,Z 540.569,A -85,B 0,C 180,E1 -23853,E2 -23853} C_VEL
LIN {X 0,Y 147.891,Z 540.765,A -85,B 0,C 180,E1 -23858.195,E2 -23858.195} C_VEL
LIN {X 0,Y 148.325,Z 540.315,A -85,B 0,C 180,E1 -23860.924,E2 -23860.924} C_VEL
LIN {X 0,Y 149.063,Z 539.448,A -85,B 0,C 180,E1 -23863.633,E2 -23863.633} C_VEL
LIN {X 0,Y 150.065,Z 538.172,A -85,B 0,C 180,E1 -23866.318,E2 -23866.318} C_VEL
LIN {X 0,Y 153.237,Z 534.43,A -85,B 0,C 180,E1 -23871.523,E2 -23871.523} C_VEL
LIN {X 0,Y 156.427,Z 530.426,A -85,B 0,C 180,E1 -23875.264,E2 -23875.264} C_VEL
LIN {X 0,Y 160.783,Z 524.312,A -85,B 0,C 180,E1 -23879.454,E2 -23879.454} C_VEL
LIN {X 0,Y 165.263,Z 517.662,A -85,B 0,C 180,E1 -23882.832,E2 -23882.832} C_VEL
LIN {X 0,Y 170.449,Z 509.436,A -85,B 0,C 180,E1 -23885.982,E2 -23885.982} C_VEL
LIN {X 0,Y 175.181,Z 501.04,A -85,B 0,C 180,E1 -23888.448,E2 -23888.448} C_VEL
LIN {X 0,Y 179.727,Z 491.874,A -85,B 0,C 180,E1 -23890.547,E2 -23890.547} C_VEL
LIN {X 0,Y 184.008,Z 481.923,A -85,B 0,C 180,E1 -23892.31,E2 -23892.31} C_VEL
LIN {X 0,Y 187.855,Z 471.132,A -85,B 0,C 180,E1 -23893.796,E2 -23893.796} C_VEL
LIN {X 0,Y 191.511,Z 458.609,A -85,B 0,C 180,E1 -23895.048,E2 -23895.048} C_VEL
LIN {X 0,Y 194.2,Z 446.068,A -85,B 0,C 180,E1 -23895.935,E2 -23895.935} C_VEL
LIN {X 0,Y 195.984,Z 432.25,A -85,B 0,C 180,E1 -23896.573,E2 -23896.573} C_VEL
LIN {X 0,Y 198.091,Z 402.881,A -85,B 0,C 180,E1 -23897.511,E2 -23897.511} C_VEL
LIN {X 0,Y 193.64,Z 391.305,A -85,B 0,C 180,E1 -23899.892,E2 -23899.892} C_VEL
LIN {X 0,Y 188.726,Z 380.505,A -85,B 0,C 180,E1 -23902.7,E2 -23902.7} C_VEL
LIN {X 0,Y 183.924,Z 371.224,A -85,B 0,C 180,E1 -23905.734,E2 -23905.734} C_VEL
LIN {X 0,Y 180.751,Z 365.728,A -85,B 0,C 180,E1 -23907.951,E2 -23907.951} C_VEL
LIN {X 0,Y 178.231,Z 361.307,A -85,B 0,C 180,E1 -23909.9,E2 -23909.9} C_VEL
LIN {X 0,Y 174.924,Z 356.03,A -85,B 0,C 180,E1 -23912.73,E2 -23912.73} C_VEL
LIN {X 0,Y 171.027,Z 350.019,A -85,B 0,C 180,E1 -23916.702,E2 -23916.702} C_VEL
LIN {X 0,Y 168.239,Z 347.243,A -85,B 0,C 180,E1 -23920.04,E2 -23920.04} C_VEL
LIN {X 0,Y 167.05,Z 344.79,A -85,B 0,C 180,E1 -23921.965,E2 -23921.965} C_VEL
LIN {X 0,Y 164.185,Z 342.639,A -85,B 0,C 180,E1 -23927.429,E2 -23927.429} C_VEL
LIN {X 0,Y 163.012,Z 339.058,A -85,B 0,C 180,E1 -23933.191,E2 -23933.191} C_VEL
LIN {X 0,Y 163.241,Z 339.054,A -85,B 0,C 180,E1 -23939.846,E2 -23939.846} C_VEL
LIN {X 0,Y 163.973,Z 341.976,A -85,B 0,C 180,E1 -23943.533,E2 -23943.533} C_VEL
LIN {X 0,Y 166.764,Z 344.429,A -85,B 0,C 180,E1 -23949.247,E2 -23949.247} C_VEL
LIN {X 0,Y 167.326,Z 344.908,A -85,B 0,C 180,E1 -23950.109,E2 -23950.109} C_VEL
LIN {X 0,Y 168.977,Z 348.051,A -85,B 0,C 180,E1 -23952.613,E2 -23952.613} C_VEL
LIN {X 0,Y 171.541,Z 350.502,A -85,B 0,C 180,E1 -23955.521,E2 -23955.521} C_VEL
LIN {X 0,Y 173.79,Z 353.935,A -85,B 0,C 180,E1 -23957.847,E2 -23957.847} C_VEL
LIN {X 0,Y 175.438,Z 355.647,A -85,B 0,C 180,E1 -23959.299,E2 -23959.299} C_VEL
LIN {X 0,Y 178.236,Z 359.483,A -85,B 0,C 180,E1 -23961.62,E2 -23961.62} C_VEL
LIN {X 0,Y 182.349,Z 365.413,A -85,B 0,C 180,E1 -23964.629,E2 -23964.629} C_VEL
LIN {X 0,Y 186.884,Z 372.127,A -85,B 0,C 180,E1 -23967.526,E2 -23967.526} C_VEL
LIN {X 0,Y 192.449,Z 381.324,A -85,B 0,C 180,E1 -23970.673,E2 -23970.673} C_VEL
LIN {X 0,Y 197.834,Z 391.35,A -85,B 0,C 180,E1 -23973.413,E2 -23973.413} C_VEL
LIN {X 0,Y 198.739,Z 393.142,A -85,B 0,C 180,E1 -23973.848,E2 -23973.848} C_VEL
LIN {X 0,Y 197.204,Z 415.476,A -85,B 0,C 180,E1 -23974.568,E2 -23974.568} C_VEL
LIN {X 0,Y 195.838,Z 429.114,A -85,B 0,C 180,E1 -23975.092,E2 -23975.092} C_VEL
LIN {X 0,Y 193.893,Z 440.961,A -85,B 0,C 180,E1 -23975.867,E2 -23975.867} C_VEL
LIN {X 0,Y 190.892,Z 453.515,A -85,B 0,C 180,E1 -23977.019,E2 -23977.019} C_VEL
LIN {X 0,Y 187.236,Z 464.978,A -85,B 0,C 180,E1 -23978.415,E2 -23978.415} C_VEL
LIN {X 0,Y 183.156,Z 475.845,A -85,B 0,C 180,E1 -23980.232,E2 -23980.232} C_VEL
LIN {X 0,Y 178.696,Z 486.008,A -85,B 0,C 180,E1 -23982.49,E2 -23982.49} C_VEL
LIN {X 0,Y 173.956,Z 495.01,A -85,B 0,C 180,E1 -23985.009,E2 -23985.009} C_VEL
LIN {X 0,Y 169.592,Z 502.402,A -85,B 0,C 180,E1 -23987.671,E2 -23987.671} C_VEL
LIN {X 0,Y 164.818,Z 509.632,A -85,B 0,C 180,E1 -23991.029,E2 -23991.029} C_VEL
LIN {X 0,Y 161.219,Z 514.477,A -85,B 0,C 180,E1 -23993.951,E2 -23993.951} C_VEL
LIN {X 0,Y 157.427,Z 519.148,A -85,B 0,C 180,E1 -23997.609,E2 -23997.609} C_VEL
LIN {X 0,Y 155.273,Z 521.615,A -85,B 0,C 180,E1 -24000.142,E2 -24000.142} C_VEL
LIN {X 0,Y 153.359,Z 523.602,A -85,B 0,C 180,E1 -24002.726,E2 -24002.726} C_VEL
LIN {X 0,Y 151.777,Z 525.163,A -85,B 0,C 180,E1 -24005.373,E2 -24005.373} C_VEL
LIN {X 0,Y 149.752,Z 526.798,A -85,B 0,C 180,E1 -24009.824,E2 -24009.824} C_VEL
LIN {X 0,Y 148.638,Z 527.277,A -85,B 0,C 180,E1 -24013.521,E2 -24013.521} C_VEL
LIN {X 0,Y 148.03,Z 527.191,A -85,B 0,C 180,E1 -24016.27,E2 -24016.27} C_VEL
LIN {X 0,Y 147.758,Z 526.687,A -85,B 0,C 180,E1 -24019.034,E2 -24019.034} C_VEL
LIN {X 0,Y 147.734,Z 525.758,A -85,B 0,C 180,E1 -24021.797,E2 -24021.797} C_VEL
LIN {X 0,Y 148.078,Z 523.995,A -85,B 0,C 180,E1 -24025.351,E2 -24025.351} C_VEL
LIN {X 0,Y 148.667,Z 520.55,A -85,B 0,C 180,E1 -24030.002,E2 -24030.002} C_VEL
LIN {X 0,Y 149.832,Z 516.423,A -85,B 0,C 180,E1 -24034.036,E2 -24034.036} C_VEL
LIN {X 0,Y 151.802,Z 510.133,A -85,B 0,C 180,E1 -24038.656,E2 -24038.656} C_VEL
LIN {X 0,Y 154.098,Z 503.294,A -85,B 0,C 180,E1 -24042.513,E2 -24042.513} C_VEL
LIN {X 0,Y 156.976,Z 494.738,A -85,B 0,C 180,E1 -24046.251,E2 -24046.251} C_VEL
LIN {X 0,Y 159.887,Z 485.95,A -85,B 0,C 180,E1 -24049.25,E2 -24049.25} C_VEL
LIN {X 0,Y 163.127,Z 475.141,A -85,B 0,C 180,E1 -24052.148,E2 -24052.148} C_VEL
LIN {X 0,Y 165.998,Z 464.234,A -85,B 0,C 180,E1 -24054.382,E2 -24054.382} C_VEL
LIN {X 0,Y 168.453,Z 452.081,A -85,B 0,C 180,E1 -24056.315,E2 -24056.315} C_VEL
LIN {X 0,Y 170.563,Z 439.26,A -85,B 0,C 180,E1 -24057.785,E2 -24057.785} C_VEL
LIN {X 0,Y 171.987,Z 426.315,A -85,B 0,C 180,E1 -24058.78,E2 -24058.78} C_VEL
LIN {X 0,Y 173.086,Z 408.711,A -85,B 0,C 180,E1 -24059.549,E2 -24059.549} C_VEL
LIN {X 0,Y 175.128,Z 370.869,A -85,B 0,C 180,E1 -24060.957,E2 -24060.957} C_VEL
LIN {X 0,Y 168.244,Z 356.348,A -85,B 0,C 180,E1 -24063.471,E2 -24063.471} C_VEL
LIN {X 0,Y 160.56,Z 343.017,A -85,B 0,C 180,E1 -24066.483,E2 -24066.483} C_VEL
LIN {X 0,Y 155.44,Z 335.453,A -85,B 0,C 180,E1 -24068.662,E2 -24068.662} C_VEL
LIN {X 0,Y 153.327,Z 332.094,A -85,B 0,C 180,E1 -24069.644,E2 -24069.644} C_VEL
LIN {X 0,Y 150.898,Z 329.176,A -85,B 0,C 180,E1 -24070.764,E2 -24070.764} C_VEL
LIN {X 0,Y 150.136,Z 326.766,A -85,B 0,C 180,E1 -24071.33,E2 -24071.33} C_VEL
LIN {X 0,Y 150.131,Z 326.774,A -85,B 0,C 180,E1 -24075.396,E2 -24075.396} C_VEL
LIN {X 0,Y 150.14,Z 326.765,A -85,B 0,C 180,E1 -24079.054,E2 -24079.054} C_VEL
LIN {X 0,Y 150.18,Z 326.769,A -85,B 0,C 180,E1 -24082.71,E2 -24082.71} C_VEL
LIN {X 0,Y 150.213,Z 326.757,A -85,B 0,C 180,E1 -24087.373,E2 -24087.373} C_VEL
LIN {X 0,Y 150.244,Z 326.749,A -85,B 0,C 180,E1 -24092.723,E2 -24092.723} C_VEL
LIN {X 0,Y 150.354,Z 326.755,A -85,B 0,C 180,E1 -24099.21,E2 -24099.21} C_VEL
LIN {X 0,Y 150.351,Z 326.725,A -85,B 0,C 180,E1 -24103.711,E2 -24103.711} C_VEL
LIN {X 0,Y 150.613,Z 326.721,A -85,B 0,C 180,E1 -24109.242,E2 -24109.242} C_VEL
LIN {X 0,Y 150.703,Z 326.703,A -85,B 0,C 180,E1 -24111.957,E2 -24111.957} C_VEL
LIN {X 0,Y 151.201,Z 326.648,A -85,B 0,C 180,E1 -24119.999,E2 -24119.999} C_VEL
LIN {X 0,Y 150.685,Z 326.689,A -85,B 0,C 180,E1 -24128.043,E2 -24128.043} C_VEL
LIN {X 0,Y 150.578,Z 326.728,A -85,B 0,C 180,E1 -24131.429,E2 -24131.429} C_VEL
LIN {X 0,Y 150.325,Z 326.761,A -85,B 0,C 180,E1 -24136.29,E2 -24136.29} C_VEL
LIN {X 0,Y 150.288,Z 326.767,A -85,B 0,C 180,E1 -24140.723,E2 -24140.723} C_VEL
LIN {X 0,Y 150.242,Z 326.768,A -85,B 0,C 180,E1 -24147.276,E2 -24147.276} C_VEL
LIN {X 0,Y 150.211,Z 326.777,A -85,B 0,C 180,E1 -24152.627,E2 -24152.627} C_VEL
LIN {X 0,Y 150.17,Z 326.781,A -85,B 0,C 180,E1 -24158.967,E2 -24158.967} C_VEL
LIN {X 0,Y 150.185,Z 327.053,A -85,B 0,C 180,E1 -24159.178,E2 -24159.178} C_VEL
LIN {X 0,Y 151.295,Z 329.84,A -85,B 0,C 180,E1 -24159.804,E2 -24159.804} C_VEL
LIN {X 0,Y 153.404,Z 332.192,A -85,B 0,C 180,E1 -24160.76,E2 -24160.76} C_VEL
LIN {X 0,Y 158.895,Z 341.918,A -85,B 0,C 180,E1 -24163.28,E2 -24163.28} C_VEL
LIN {X 0,Y 164.83,Z 353.805,A -85,B 0,C 180,E1 -24165.795,E2 -24165.795} C_VEL
LIN {X 0,Y 170.14,Z 366.726,A -85,B 0,C 180,E1 -24167.95,E2 -24167.95} C_VEL
LIN {X 0,Y 172.573,Z 374.25,A -85,B 0,C 180,E1 -24168.956,E2 -24168.956} C_VEL
LIN {X 0,Y 174.054,Z 394.935,A -85,B 0,C 180,E1 -24170.354,E2 -24170.354} C_VEL
LIN {X 0,Y 171.731,Z 437.077,A -85,B 0,C 180,E1 -24171.991,E2 -24171.991} C_VEL
LIN {X 0,Y 170.156,Z 450.649,A -85,B 0,C 180,E1 -24172.93,E2 -24172.93} C_VEL
LIN {X 0,Y 168.041,Z 462.676,A -85,B 0,C 180,E1 -24174.158,E2 -24174.158} C_VEL
LIN {X 0,Y 165.528,Z 474.033,A -85,B 0,C 180,E1 -24175.765,E2 -24175.765} C_VEL
LIN {X 0,Y 162.362,Z 485.748,A -85,B 0,C 180,E1 -24177.976,E2 -24177.976} C_VEL
LIN {X 0,Y 159.277,Z 496.305,A -85,B 0,C 180,E1 -24180.599,E2 -24180.599} C_VEL
LIN {X 0,Y 156.57,Z 504.93,A -85,B 0,C 180,E1 -24183.327,E2 -24183.327} C_VEL
LIN {X 0,Y 153.934,Z 512.87,A -85,B 0,C 180,E1 -24186.452,E2 -24186.452} C_VEL
LIN {X 0,Y 151.531,Z 520.622,A -85,B 0,C 180,E1 -24190.349,E2 -24190.349} C_VEL
LIN {X 0,Y 149.352,Z 527.747,A -85,B 0,C 180,E1 -24194.999,E2 -24194.999} C_VEL
LIN {X 0,Y 148.314,Z 532.478,A -85,B 0,C 180,E1 -24199.072,E2 -24199.072} C_VEL
LIN {X 0,Y 147.984,Z 534.776,A -85,B 0,C 180,E1 -24201.558,E2 -24201.558} C_VEL
LIN {X 0,Y 147.171,Z 536.515,A -85,B 0,C 180,E1 -24203.729,E2 -24203.729} C_VEL
LIN {X 0,Y 145.539,Z 537.889,A -85,B 0,C 180,E1 -24205.905,E2 -24205.905} C_VEL
LIN {X 0,Y 141.832,Z 539.661,A -85,B 0,C 180,E1 -24210.422,E2 -24210.422} C_VEL
LIN {X 0,Y 140.66,Z 540.25,A -85,B 0,C 180,E1 -24213.634,E2 -24213.634} C_VEL
LIN {X 0,Y 140.837,Z 540.445,A -85,B 0,C 180,E1 -24218.608,E2 -24218.608} C_VEL
LIN {X 0,Y 142.145,Z 539.195,A -85,B 0,C 180,E1 -24224.311,E2 -24224.311} C_VEL
LIN {X 0,Y 143.23,Z 537.943,A -85,B 0,C 180,E1 -24227.12,E2 -24227.12} C_VEL
LIN {X 0,Y 146.615,Z 534.25,A -85,B 0,C 180,E1 -24232.547,E2 -24232.547} C_VEL
LIN {X 0,Y 150.004,Z 530.296,A -85,B 0,C 180,E1 -24236.427,E2 -24236.427} C_VEL
LIN {X 0,Y 153.917,Z 525.232,A -85,B 0,C 180,E1 -24240.148,E2 -24240.148} C_VEL
LIN {X 0,Y 158.507,Z 518.905,A -85,B 0,C 180,E1 -24243.656,E2 -24243.656} C_VEL
LIN {X 0,Y 163.834,Z 511.012,A -85,B 0,C 180,E1 -24246.908,E2 -24246.908} C_VEL
LIN {X 0,Y 168.652,Z 502.996,A -85,B 0,C 180,E1 -24249.454,E2 -24249.454} C_VEL
LIN {X 0,Y 173.35,Z 494.305,A -85,B 0,C 180,E1 -24251.595,E2 -24251.595} C_VEL
LIN {X 0,Y 177.705,Z 484.985,A -85,B 0,C 180,E1 -24253.404,E2 -24253.404} C_VEL
LIN {X 0,Y 182.249,Z 473.468,A -85,B 0,C 180,E1 -24255.118,E2 -24255.118} C_VEL
LIN {X 0,Y 186.076,Z 461.548,A -85,B 0,C 180,E1 -24256.403,E2 -24256.403} C_VEL
LIN {X 0,Y 189.165,Z 448.501,A -85,B 0,C 180,E1 -24257.41,E2 -24257.41} C_VEL
LIN {X 0,Y 191.224,Z 435.168,A -85,B 0,C 180,E1 -24258.109,E2 -24258.109} C_VEL
LIN {X 0,Y 193.555,Z 405.255,A -85,B 0,C 180,E1 -24259.075,E2 -24259.075} C_VEL
LIN {X 0,Y 189.353,Z 394.224,A -85,B 0,C 180,E1 -24261.505,E2 -24261.505} C_VEL
LIN {X 0,Y 184.671,Z 383.84,A -85,B 0,C 180,E1 -24264.408,E2 -24264.408} C_VEL
LIN {X 0,Y 180.565,Z 375.761,A -85,B 0,C 180,E1 -24267.237,E2 -24267.237} C_VEL
LIN {X 0,Y 176.366,Z 367.949,A -85,B 0,C 180,E1 -24270.537,E2 -24270.537} C_VEL
LIN {X 0,Y 172.951,Z 362.282,A -85,B 0,C 180,E1 -24273.616,E2 -24273.616} C_VEL
LIN {X 0,Y 169.602,Z 356.844,A -85,B 0,C 180,E1 -24277.221,E2 -24277.221} C_VEL
LIN {X 0,Y 166.766,Z 353.802,A -85,B 0,C 180,E1 -24280.821,E2 -24280.821} C_VEL
LIN {X 0,Y 165.652,Z 351.621,A -85,B 0,C 180,E1 -24282.724,E2 -24282.724} C_VEL
LIN {X 0,Y 163.043,Z 349.34,A -85,B 0,C 180,E1 -24288.186,E2 -24288.186} C_VEL
LIN {X 0,Y 162.095,Z 346.068,A -85,B 0,C 180,E1 -24293.611,E2 -24293.611} C_VEL
LIN {X 0,Y 162.303,Z 346.152,A -85,B 0,C 180,E1 -24299.535,E2 -24299.535} C_VEL
LIN {X 0,Y 163.015,Z 349.03,A -85,B 0,C 180,E1 -24303.322,E2 -24303.322} C_VEL
LIN {X 0,Y 165.96,Z 351.65,A -85,B 0,C 180,E1 -24309.407,E2 -24309.407} C_VEL
LIN {X 0,Y 167.867,Z 355.14,A -85,B 0,C 180,E1 -24312.391,E2 -24312.391} C_VEL
LIN {X 0,Y 169.931,Z 357.188,A -85,B 0,C 180,E1 -24314.828,E2 -24314.828} C_VEL
LIN {X 0,Y 172.362,Z 360.792,A -85,B 0,C 180,E1 -24317.425,E2 -24317.425} C_VEL
LIN {X 0,Y 173.688,Z 362.389,A -85,B 0,C 180,E1 -24318.658,E2 -24318.658} C_VEL
LIN {X 0,Y 177.181,Z 367.397,A -85,B 0,C 180,E1 -24321.64,E2 -24321.64} C_VEL
LIN {X 0,Y 180.319,Z 372.041,A -85,B 0,C 180,E1 -24323.996,E2 -24323.996} C_VEL
LIN {X 0,Y 185.633,Z 380.349,A -85,B 0,C 180,E1 -24327.498,E2 -24327.498} C_VEL
LIN {X 0,Y 190.926,Z 389.675,A -85,B 0,C 180,E1 -24330.561,E2 -24330.561} C_VEL
LIN {X 0,Y 194.274,Z 396.297,A -85,B 0,C 180,E1 -24332.346,E2 -24332.346} C_VEL
LIN {X 0,Y 191.737,Z 426.013,A -85,B 0,C 180,E1 -24333.283,E2 -24333.283} C_VEL
LIN {X 0,Y 189.819,Z 438.759,A -85,B 0,C 180,E1 -24334.047,E2 -24334.047} C_VEL
LIN {X 0,Y 186.976,Z 451.462,A -85,B 0,C 180,E1 -24335.164,E2 -24335.164} C_VEL
LIN {X 0,Y 183.441,Z 462.606,A -85,B 0,C 180,E1 -24336.435,E2 -24336.435} C_VEL
LIN {X 0,Y 178.979,Z 474.223,A -85,B 0,C 180,E1 -24338.25,E2 -24338.25} C_VEL
LIN {X 0,Y 174.389,Z 484.657,A -85,B 0,C 180,E1 -24340.479,E2 -24340.479} C_VEL
LIN {X 0,Y 168.924,Z 494.77,A -85,B 0,C 180,E1 -24343.277,E2 -24343.277} C_VEL
LIN {X 0,Y 163.408,Z 503.623,A -85,B 0,C 180,E1 -24346.519,E2 -24346.519} C_VEL
LIN {X 0,Y 158.442,Z 510.634,A -85,B 0,C 180,E1 -24349.973,E2 -24349.973} C_VEL
LIN {X 0,Y 153.99,Z 516.205,A -85,B 0,C 180,E1 -24353.61,E2 -24353.61} C_VEL
LIN {X 0,Y 150.206,Z 520.486,A -85,B 0,C 180,E1 -24357.375,E2 -24357.375} C_VEL
LIN {X 0,Y 146.946,Z 523.78,A -85,B 0,C 180,E1 -24361.43,E2 -24361.43} C_VEL
LIN {X 0,Y 145.198,Z 525.372,A -85,B 0,C 180,E1 -24364.177,E2 -24364.177} C_VEL
LIN {X 0,Y 142.825,Z 527.169,A -85,B 0,C 180,E1 -24369.22,E2 -24369.22} C_VEL
LIN {X 0,Y 141.729,Z 527.599,A -85,B 0,C 180,E1 -24372.693,E2 -24372.693} C_VEL
LIN {X 0,Y 140.693,Z 527.086,A -85,B 0,C 180,E1 -24378.476,E2 -24378.476} C_VEL
LIN {X 0,Y 140.629,Z 526.19,A -85,B 0,C 180,E1 -24381.379,E2 -24381.379} C_VEL
LIN {X 0,Y 140.995,Z 524.236,A -85,B 0,C 180,E1 -24385.514,E2 -24385.514} C_VEL
LIN {X 0,Y 141.58,Z 521.094,A -85,B 0,C 180,E1 -24390.002,E2 -24390.002} C_VEL
LIN {X 0,Y 142.747,Z 517.033,A -85,B 0,C 180,E1 -24394.237,E2 -24394.237} C_VEL
LIN {X 0,Y 144.817,Z 510.81,A -85,B 0,C 180,E1 -24399.077,E2 -24399.077} C_VEL
LIN {X 0,Y 147.186,Z 504.05,A -85,B 0,C 180,E1 -24403.111,E2 -24403.111} C_VEL
LIN {X 0,Y 150.205,Z 495.629,A -85,B 0,C 180,E1 -24407.006,E2 -24407.006} C_VEL
LIN {X 0,Y 153.218,Z 486.955,A -85,B 0,C 180,E1 -24410.124,E2 -24410.124} C_VEL
LIN {X 0,Y 156.608,Z 476.282,A -85,B 0,C 180,E1 -24413.122,E2 -24413.122} C_VEL
LIN {X 0,Y 159.583,Z 465.643,A -85,B 0,C 180,E1 -24415.43,E2 -24415.43} C_VEL
LIN {X 0,Y 162.167,Z 453.78,A -85,B 0,C 180,E1 -24417.419,E2 -24417.419} C_VEL
LIN {X 0,Y 164.379,Z 441.412,A -85,B 0,C 180,E1 -24418.927,E2 -24418.927} C_VEL
LIN {X 0,Y 165.97,Z 428.631,A -85,B 0,C 180,E1 -24420.015,E2 -24420.015} C_VEL
LIN {X 0,Y 167.019,Z 414.062,A -85,B 0,C 180,E1 -24420.73,E2 -24420.73} C_VEL
LIN {X 0,Y 169.331,Z 373,A -85,B 0,C 180,E1 -24422.295,E2 -24422.295} C_VEL
LIN {X 0,Y 163.099,Z 359.799,A -85,B 0,C 180,E1 -24424.739,E2 -24424.739} C_VEL
LIN {X 0,Y 156.169,Z 347.661,A -85,B 0,C 180,E1 -24427.648,E2 -24427.648} C_VEL
LIN {X 0,Y 151.092,Z 340.064,A -85,B 0,C 180,E1 -24429.962,E2 -24429.962} C_VEL
LIN {X 0,Y 148.851,Z 336.716,A -85,B 0,C 180,E1 -24431.064,E2 -24431.064} C_VEL
LIN {X 0,Y 146.521,Z 333.212,A -85,B 0,C 180,E1 -24432.271,E2 -24432.271} C_VEL
LIN {X 0,Y 143.922,Z 330.282,A -85,B 0,C 180,E1 -24433.626,E2 -24433.626} C_VEL
LIN {X 0,Y 143.084,Z 327.66,A -85,B 0,C 180,E1 -24434.252,E2 -24434.252} C_VEL
LIN {X 0,Y 143.056,Z 327.659,A -85,B 0,C 180,E1 -24440.307,E2 -24440.307} C_VEL
LIN {X 0,Y 143.143,Z 327.63,A -85,B 0,C 180,E1 -24446.584,E2 -24446.584} C_VEL
LIN {X 0,Y 143.188,Z 327.635,A -85,B 0,C 180,E1 -24452.069,E2 -24452.069} C_VEL
LIN {X 0,Y 143.28,Z 327.636,A -85,B 0,C 180,E1 -24458.749,E2 -24458.749} C_VEL
LIN {X 0,Y 143.296,Z 327.609,A -85,B 0,C 180,E1 -24462.885,E2 -24462.885} C_VEL
LIN {X 0,Y 143.539,Z 327.6,A -85,B 0,C 180,E1 -24468.705,E2 -24468.705} C_VEL
LIN {X 0,Y 143.625,Z 327.587,A -85,B 0,C 180,E1 -24471.558,E2 -24471.558} C_VEL
LIN {X 0,Y 144.16,Z 327.525,A -85,B 0,C 180,E1 -24479.999,E2 -24479.999} C_VEL
LIN {X 0,Y 143.611,Z 327.572,A -85,B 0,C 180,E1 -24488.442,E2 -24488.442} C_VEL
LIN {X 0,Y 143.504,Z 327.609,A -85,B 0,C 180,E1 -24491.618,E2 -24491.618} C_VEL
LIN {X 0,Y 143.263,Z 327.638,A -85,B 0,C 180,E1 -24497.117,E2 -24497.117} C_VEL
LIN {X 0,Y 143.226,Z 327.645,A -85,B 0,C 180,E1 -24501.197,E2 -24501.197} C_VEL
LIN {X 0,Y 143.186,Z 327.648,A -85,B 0,C 180,E1 -24507.93,E2 -24507.93} C_VEL
LIN {X 0,Y 143.141,Z 327.658,A -85,B 0,C 180,E1 -24513.415,E2 -24513.415} C_VEL
LIN {X 0,Y 143.101,Z 327.687,A -85,B 0,C 180,E1 -24516.168,E2 -24516.168} C_VEL
LIN {X 0,Y 144,Z 330.281,A -85,B 0,C 180,E1 -24516.774,E2 -24516.774} C_VEL
LIN {X 0,Y 146.123,Z 332.608,A -85,B 0,C 180,E1 -24517.88,E2 -24517.88} C_VEL
LIN {X 0,Y 148.809,Z 336.666,A -85,B 0,C 180,E1 -24519.283,E2 -24519.283} C_VEL
LIN {X 0,Y 150.421,Z 339.069,A -85,B 0,C 180,E1 -24520.082,E2 -24520.082} C_VEL
LIN {X 0,Y 154.683,Z 346.781,A -85,B 0,C 180,E1 -24522.152,E2 -24522.152} C_VEL
LIN {X 0,Y 160.025,Z 357.757,A -85,B 0,C 180,E1 -24524.579,E2 -24524.579} C_VEL
LIN {X 0,Y 165.039,Z 370.289,A -85,B 0,C 180,E1 -24526.766,E2 -24526.766} C_VEL
LIN {X 0,Y 166.933,Z 375.889,A -85,B 0,C 180,E1 -24527.589,E2 -24527.589} C_VEL
LIN {X 0,Y 168.295,Z 395.519,A -85,B 0,C 180,E1 -24528.985,E2 -24528.985} C_VEL
LIN {X 0,Y 165.875,Z 436.983,A -85,B 0,C 180,E1 -24530.636,E2 -24530.636} C_VEL
LIN {X 0,Y 164.175,Z 450.877,A -85,B 0,C 180,E1 -24531.63,E2 -24531.63} C_VEL
LIN {X 0,Y 161.87,Z 463.29,A -85,B 0,C 180,E1 -24532.955,E2 -24532.955} C_VEL
LIN {X 0,Y 158.815,Z 475.984,A -85,B 0,C 180,E1 -24534.878,E2 -24534.878} C_VEL
LIN {X 0,Y 155.623,Z 487.293,A -85,B 0,C 180,E1 -24537.183,E2 -24537.183} C_VEL
LIN {X 0,Y 152.373,Z 497.456,A -85,B 0,C 180,E1 -24539.893,E2 -24539.893} C_VEL
LIN {X 0,Y 149.02,Z 507.473,A -85,B 0,C 180,E1 -24543.382,E2 -24543.382} C_VEL
LIN {X 0,Y 146.928,Z 513.643,A -85,B 0,C 180,E1 -24546.063,E2 -24546.063} C_VEL
LIN {X 0,Y 144.438,Z 521.103,A -85,B 0,C 180,E1 -24550.085,E2 -24550.085} C_VEL
LIN {X 0,Y 142.445,Z 527.156,A -85,B 0,C 180,E1 -24554.253,E2 -24554.253} C_VEL
LIN {X 0,Y 141.319,Z 531.944,A -85,B 0,C 180,E1 -24558.524,E2 -24558.524} C_VEL
LIN {X 0,Y 140.785,Z 535.59,A -85,B 0,C 180,E1 -24562.829,E2 -24562.829} C_VEL
LIN {X 0,Y 140.775,Z 538.199,A -85,B 0,C 180,E1 -24567.137,E2 -24567.137} C_VEL
LIN {X 0,Y 140.917,Z 539.413,A -85,B 0,C 180,E1 -24569.998,E2 -24569.998} C_VEL
LIN {X 0,Y 140.66,Z 540.25,A -85,B 0,C 180,E1 -24573.634,E2 -24573.634} C_VEL
LIN {X 0,Y 139.991,Z 540.486,A -85,B 0,C 180,E1 -24576.03,E2 -24576.03} C_VEL
LIN {X 0,Y 137.513,Z 540.187,A -85,B 0,C 180,E1 -24579.997,E2 -24579.997} C_VEL
LIN {X 0,Y 135.8,Z 539.469,A -85,B 0,C 180,E1 -24583.253,E2 -24583.253} C_VEL
LIN {X 0,Y 135.559,Z 538.674,A -85,B 0,C 180,E1 -24585.736,E2 -24585.736} C_VEL
LIN {X 0,Y 135.794,Z 538.316,A -85,B 0,C 180,E1 -24586.555,E2 -24586.555} C_VEL
LIN {X 0,Y 139.046,Z 535.154,A -85,B 0,C 180,E1 -24592.275,E2 -24592.275} C_VEL
LIN {X 0,Y 142.394,Z 531.605,A -85,B 0,C 180,E1 -24596.37,E2 -24596.37} C_VEL
LIN {X 0,Y 146.738,Z 526.457,A -85,B 0,C 180,E1 -24600.646,E2 -24600.646} C_VEL
LIN {X 0,Y 151.775,Z 520.018,A -85,B 0,C 180,E1 -24604.556,E2 -24604.556} C_VEL
LIN {X 0,Y 157.222,Z 512.519,A -85,B 0,C 180,E1 -24607.924,E2 -24607.924} C_VEL
LIN {X 0,Y 162.206,Z 504.889,A -85,B 0,C 180,E1 -24610.533,E2 -24610.533} C_VEL
LIN {X 0,Y 167.553,Z 495.657,A -85,B 0,C 180,E1 -24612.967,E2 -24612.967} C_VEL
LIN {X 0,Y 172.629,Z 485.401,A -85,B 0,C 180,E1 -24615.019,E2 -24615.019} C_VEL
LIN {X 0,Y 177.331,Z 474.051,A -85,B 0,C 180,E1 -24616.737,E2 -24616.737} C_VEL
LIN {X 0,Y 181.014,Z 463.338,A -85,B 0,C 180,E1 -24617.927,E2 -24617.927} C_VEL
LIN {X 0,Y 184.278,Z 450.922,A -85,B 0,C 180,E1 -24618.952,E2 -24618.952} C_VEL
LIN {X 0,Y 186.597,Z 437.635,A -85,B 0,C 180,E1 -24619.702,E2 -24619.702} C_VEL
LIN {X 0,Y 188.594,Z 416.531,A -85,B 0,C 180,E1 -24620.385,E2 -24620.385} C_VEL
LIN {X 0,Y 189.22,Z 407.894,A -85,B 0,C 180,E1 -24620.675,E2 -24620.675} C_VEL
LIN {X 0,Y 185.352,Z 397.548,A -85,B 0,C 180,E1 -24623.1,E2 -24623.1} C_VEL
LIN {X 0,Y 180.756,Z 387.096,A -85,B 0,C 180,E1 -24626.224,E2 -24626.224} C_VEL
LIN {X 0,Y 176.46,Z 378.445,A -85,B 0,C 180,E1 -24629.517,E2 -24629.517} C_VEL
LIN {X 0,Y 173.061,Z 372.168,A -85,B 0,C 180,E1 -24632.498,E2 -24632.498} C_VEL
LIN {X 0,Y 170.59,Z 367.9,A -85,B 0,C 180,E1 -24634.963,E2 -24634.963} C_VEL
LIN {X 0,Y 168.071,Z 363.516,A -85,B 0,C 180,E1 -24637.893,E2 -24637.893} C_VEL
LIN {X 0,Y 165.368,Z 360.438,A -85,B 0,C 180,E1 -24641.545,E2 -24641.545} C_VEL
LIN {X 0,Y 164.44,Z 358.534,A -85,B 0,C 180,E1 -24643.233,E2 -24643.233} C_VEL
LIN {X 0,Y 161.895,Z 356.042,A -85,B 0,C 180,E1 -24649.052,E2 -24649.052} C_VEL
LIN {X 0,Y 161.214,Z 353.231,A -85,B 0,C 180,E1 -24653.587,E2 -24653.587} C_VEL
LIN {X 0,Y 161.364,Z 353.09,A -85,B 0,C 180,E1 -24659.065,E2 -24659.065} C_VEL
LIN {X 0,Y 161.971,Z 355.894,A -85,B 0,C 180,E1 -24662.799,E2 -24662.799} C_VEL
LIN {X 0,Y 164.722,Z 358.657,A -85,B 0,C 180,E1 -24668.898,E2 -24668.898} C_VEL
LIN {X 0,Y 166.603,Z 362.026,A -85,B 0,C 180,E1 -24671.951,E2 -24671.951} C_VEL
LIN {X 0,Y 168.374,Z 363.935,A -85,B 0,C 180,E1 -24674.157,E2 -24674.157} C_VEL
LIN {X 0,Y 171.12,Z 367.862,A -85,B 0,C 180,E1 -24677.17,E2 -24677.17} C_VEL
LIN {X 0,Y 175.057,Z 373.64,A -85,B 0,C 180,E1 -24680.778,E2 -24680.778} C_VEL
LIN {X 0,Y 178.095,Z 378.316,A -85,B 0,C 180,E1 -24683.185,E2 -24683.185} C_VEL
LIN {X 0,Y 183.09,Z 386.466,A -85,B 0,C 180,E1 -24686.657,E2 -24686.657} C_VEL
LIN {X 0,Y 188.042,Z 395.639,A -85,B 0,C 180,E1 -24689.69,E2 -24689.69} C_VEL
LIN {X 0,Y 189.814,Z 399.216,A -85,B 0,C 180,E1 -24690.7,E2 -24690.7} C_VEL
LIN {X 0,Y 187.446,Z 426.384,A -85,B 0,C 180,E1 -24691.584,E2 -24691.584} C_VEL
LIN {X 0,Y 185.322,Z 439.844,A -85,B 0,C 180,E1 -24692.402,E2 -24692.402} C_VEL
LIN {X 0,Y 182.29,Z 452.431,A -85,B 0,C 180,E1 -24693.519,E2 -24693.519} C_VEL
LIN {X 0,Y 178.051,Z 465.05,A -85,B 0,C 180,E1 -24695.014,E2 -24695.014} C_VEL
LIN {X 0,Y 173.379,Z 476.506,A -85,B 0,C 180,E1 -24696.914,E2 -24696.914} C_VEL
LIN {X 0,Y 168.191,Z 487.29,A -85,B 0,C 180,E1 -24699.375,E2 -24699.375} C_VEL
LIN {X 0,Y 163.026,Z 496.186,A -85,B 0,C 180,E1 -24701.96,E2 -24701.96} C_VEL
LIN {X 0,Y 157.415,Z 504.647,A -85,B 0,C 180,E1 -24705.219,E2 -24705.219} C_VEL
LIN {X 0,Y 152.119,Z 511.631,A -85,B 0,C 180,E1 -24708.827,E2 -24708.827} C_VEL
LIN {X 0,Y 146.779,Z 517.875,A -85,B 0,C 180,E1 -24713.238,E2 -24713.238} C_VEL
LIN {X 0,Y 142.852,Z 521.9,A -85,B 0,C 180,E1 -24717.238,E2 -24717.238} C_VEL
LIN {X 0,Y 140.628,Z 523.959,A -85,B 0,C 180,E1 -24720.018,E2 -24720.018} C_VEL
LIN {X 0,Y 138.705,Z 525.58,A -85,B 0,C 180,E1 -24722.872,E2 -24722.872} C_VEL
LIN {X 0,Y 135.921,Z 527.532,A -85,B 0,C 180,E1 -24728.55,E2 -24728.55} C_VEL
LIN {X 0,Y 134.836,Z 527.921,A -85,B 0,C 180,E1 -24731.778,E2 -24731.778} C_VEL
LIN {X 0,Y 133.656,Z 527.468,A -85,B 0,C 180,E1 -24737.86,E2 -24737.86} C_VEL
LIN {X 0,Y 133.526,Z 526.623,A -85,B 0,C 180,E1 -24740.917,E2 -24740.917} C_VEL
LIN {X 0,Y 133.921,Z 524.501,A -85,B 0,C 180,E1 -24745.649,E2 -24745.649} C_VEL
LIN {X 0,Y 134.49,Z 521.632,A -85,B 0,C 180,E1 -24750.002,E2 -24750.002} C_VEL
LIN {X 0,Y 135.665,Z 517.635,A -85,B 0,C 180,E1 -24754.459,E2 -24754.459} C_VEL
LIN {X 0,Y 137.808,Z 511.489,A -85,B 0,C 180,E1 -24759.542,E2 -24759.542} C_VEL
LIN {X 0,Y 140.296,Z 504.805,A -85,B 0,C 180,E1 -24763.767,E2 -24763.767} C_VEL
LIN {X 0,Y 143.464,Z 496.508,A -85,B 0,C 180,E1 -24767.831,E2 -24767.831} C_VEL
LIN {X 0,Y 146.591,Z 487.96,A -85,B 0,C 180,E1 -24771.076,E2 -24771.076} C_VEL
LIN {X 0,Y 150.141,Z 477.421,A -85,B 0,C 180,E1 -24774.18,E2 -24774.18} C_VEL
LIN {X 0,Y 153.258,Z 466.964,A -85,B 0,C 180,E1 -24776.56,E2 -24776.56} C_VEL
LIN {X 0,Y 155.98,Z 455.468,A -85,B 0,C 180,E1 -24778.604,E2 -24778.604} C_VEL
LIN {X 0,Y 158.267,Z 443.529,A -85,B 0,C 180,E1 -24780.157,E2 -24780.157} C_VEL
LIN {X 0,Y 160.041,Z 430.613,A -85,B 0,C 180,E1 -24781.341,E2 -24781.341} C_VEL
LIN {X 0,Y 161.065,Z 417.942,A -85,B 0,C 180,E1 -24782.07,E2 -24782.07} C_VEL
LIN {X 0,Y 163.64,Z 375.2,A -85,B 0,C 180,E1 -24783.721,E2 -24783.721} C_VEL
LIN {X 0,Y 158.066,Z 363.316,A -85,B 0,C 180,E1 -24786.076,E2 -24786.076} C_VEL
LIN {X 0,Y 151.821,Z 352.177,A -85,B 0,C 180,E1 -24788.896,E2 -24788.896} C_VEL
LIN {X 0,Y 146.778,Z 344.532,A -85,B 0,C 180,E1 -24791.365,E2 -24791.365} C_VEL
LIN {X 0,Y 142.595,Z 338.281,A -85,B 0,C 180,E1 -24793.633,E2 -24793.633} C_VEL
LIN {X 0,Y 140.22,Z 335.336,A -85,B 0,C 180,E1 -24794.982,E2 -24794.982} C_VEL
LIN {X 0,Y 139.311,Z 333.68,A -85,B 0,C 180,E1 -24795.563,E2 -24795.563} C_VEL
LIN {X 0,Y 137.078,Z 331.507,A -85,B 0,C 180,E1 -24796.897,E2 -24796.897} C_VEL
LIN {X 0,Y 136.058,Z 328.98,A -85,B 0,C 180,E1 -24797.666,E2 -24797.666} C_VEL
LIN {X 0,Y 135.987,Z 328.521,A -85,B 0,C 180,E1 -24797.788,E2 -24797.788} C_VEL
LIN {X 0,Y 136.026,Z 328.539,A -85,B 0,C 180,E1 -24801.683,E2 -24801.683} C_VEL
LIN {X 0,Y 136.057,Z 328.508,A -85,B 0,C 180,E1 -24805.742,E2 -24805.742} C_VEL
LIN {X 0,Y 136.129,Z 328.509,A -85,B 0,C 180,E1 -24812.311,E2 -24812.311} C_VEL
LIN {X 0,Y 136.246,Z 328.513,A -85,B 0,C 180,E1 -24818.832,E2 -24818.832} C_VEL
LIN {X 0,Y 136.249,Z 328.476,A -85,B 0,C 180,E1 -24825.053,E2 -24825.053} C_VEL
LIN {X 0,Y 136.431,Z 328.481,A -85,B 0,C 180,E1 -24828.177,E2 -24828.177} C_VEL
LIN {X 0,Y 136.552,Z 328.472,A -85,B 0,C 180,E1 -24831.117,E2 -24831.117} C_VEL
LIN {X 0,Y 137.117,Z 328.402,A -85,B 0,C 180,E1 -24839.999,E2 -24839.999} C_VEL
LIN {X 0,Y 136.54,Z 328.456,A -85,B 0,C 180,E1 -24848.882,E2 -24848.882} C_VEL
LIN {X 0,Y 136.419,Z 328.492,A -85,B 0,C 180,E1 -24851.892,E2 -24851.892} C_VEL
LIN {X 0,Y 136.173,Z 328.518,A -85,B 0,C 180,E1 -24858.038,E2 -24858.038} C_VEL
LIN {X 0,Y 136.152,Z 328.525,A -85,B 0,C 180,E1 -24861.694,E2 -24861.694} C_VEL
LIN {X 0,Y 136.096,Z 328.535,A -85,B 0,C 180,E1 -24868.608,E2 -24868.608} C_VEL
LIN {X 0,Y 136.14,Z 328.568,A -85,B 0,C 180,E1 -24872.712,E2 -24872.712} C_VEL
LIN {X 0,Y 136.968,Z 331.165,A -85,B 0,C 180,E1 -24873.384,E2 -24873.384} C_VEL
LIN {X 0,Y 138.905,Z 333.379,A -85,B 0,C 180,E1 -24874.576,E2 -24874.576} C_VEL
LIN {X 0,Y 139.762,Z 334.308,A -85,B 0,C 180,E1 -24875.079,E2 -24875.079} C_VEL
LIN {X 0,Y 141.897,Z 337.546,A -85,B 0,C 180,E1 -24876.355,E2 -24876.355} C_VEL
LIN {X 0,Y 143.064,Z 338.962,A -85,B 0,C 180,E1 -24876.997,E2 -24876.997} C_VEL
LIN {X 0,Y 146.569,Z 344.193,A -85,B 0,C 180,E1 -24878.891,E2 -24878.891} C_VEL
LIN {X 0,Y 152.363,Z 355.245,A -85,B 0,C 180,E1 -24881.866,E2 -24881.866} C_VEL
LIN {X 0,Y 157.443,Z 366.92,A -85,B 0,C 180,E1 -24884.307,E2 -24884.307} C_VEL
LIN {X 0,Y 161.431,Z 378.057,A -85,B 0,C 180,E1 -24886.17,E2 -24886.17} C_VEL
LIN {X 0,Y 162.605,Z 395.026,A -85,B 0,C 180,E1 -24887.452,E2 -24887.452} C_VEL
LIN {X 0,Y 160.164,Z 436.332,A -85,B 0,C 180,E1 -24889.148,E2 -24889.148} C_VEL
LIN {X 0,Y 158.496,Z 449.56,A -85,B 0,C 180,E1 -24890.089,E2 -24890.089} C_VEL
LIN {X 0,Y 156.263,Z 461.716,A -85,B 0,C 180,E1 -24891.387,E2 -24891.387} C_VEL
LIN {X 0,Y 153.524,Z 473.158,A -85,B 0,C 180,E1 -24893.068,E2 -24893.068} C_VEL
LIN {X 0,Y 150.064,Z 484.917,A -85,B 0,C 180,E1 -24895.397,E2 -24895.397} C_VEL
LIN {X 0,Y 146.589,Z 495.493,A -85,B 0,C 180,E1 -24898.169,E2 -24898.169} C_VEL
LIN {X 0,Y 143.231,Z 505.19,A -85,B 0,C 180,E1 -24901.497,E2 -24901.497} C_VEL
LIN {X 0,Y 140.247,Z 513.292,A -85,B 0,C 180,E1 -24905.06,E2 -24905.06} C_VEL
LIN {X 0,Y 137.329,Z 521.582,A -85,B 0,C 180,E1 -24909.789,E2 -24909.789} C_VEL
LIN {X 0,Y 135.579,Z 526.564,A -85,B 0,C 180,E1 -24913.433,E2 -24913.433} C_VEL
LIN {X 0,Y 134.319,Z 531.408,A -85,B 0,C 180,E1 -24917.917,E2 -24917.917} C_VEL
LIN {X 0,Y 133.724,Z 535.108,A -85,B 0,C 180,E1 -24922.448,E2 -24922.448} C_VEL
LIN {X 0,Y 133.683,Z 537.901,A -85,B 0,C 180,E1 -24927.267,E2 -24927.267} C_VEL
LIN {X 0,Y 133.82,Z 539.003,A -85,B 0,C 180,E1 -24929.998,E2 -24929.998} C_VEL
LIN {X 0,Y 133.595,Z 539.863,A -85,B 0,C 180,E1 -24933.586,E2 -24933.586} C_VEL
LIN {X 0,Y 133.808,Z 540.125,A -85,B 0,C 180,E1 -24939.064,E2 -24939.064} C_VEL
LIN {X 0,Y 135.237,Z 538.933,A -85,B 0,C 180,E1 -24945.059,E2 -24945.059} C_VEL
LIN {X 0,Y 135.794,Z 538.316,A -85,B 0,C 180,E1 -24946.555,E2 -24946.555} C_VEL
LIN {X 0,Y 136.28,Z 537.241,A -85,B 0,C 180,E1 -24948.993,E2 -24948.993} C_VEL
LIN {X 0,Y 135.94,Z 534.955,A -85,B 0,C 180,E1 -24953.054,E2 -24953.054} C_VEL
LIN {X 0,Y 135.984,Z 532.66,A -85,B 0,C 180,E1 -24956.258,E2 -24956.258} C_VEL
LIN {X 0,Y 136.96,Z 530.591,A -85,B 0,C 180,E1 -24958.548,E2 -24958.548} C_VEL
LIN {X 0,Y 137.557,Z 529.831,A -85,B 0,C 180,E1 -24959.266,E2 -24959.266} C_VEL
LIN {X 0,Y 141.763,Z 525.088,A -85,B 0,C 180,E1 -24963.045,E2 -24963.045} C_VEL
LIN {X 0,Y 146.881,Z 518.89,A -85,B 0,C 180,E1 -24966.732,E2 -24966.732} C_VEL
LIN {X 0,Y 152.712,Z 511.205,A -85,B 0,C 180,E1 -24970.111,E2 -24970.111} C_VEL
LIN {X 0,Y 159.07,Z 501.582,A -85,B 0,C 180,E1 -24973.219,E2 -24973.219} C_VEL
LIN {X 0,Y 164.702,Z 491.68,A -85,B 0,C 180,E1 -24975.619,E2 -24975.619} C_VEL
LIN {X 0,Y 170.158,Z 480.543,A -85,B 0,C 180,E1 -24977.583,E2 -24977.583} C_VEL
LIN {X 0,Y 174.44,Z 469.665,A -85,B 0,C 180,E1 -24979.059,E2 -24979.059} C_VEL
LIN {X 0,Y 178.551,Z 456.772,A -85,B 0,C 180,E1 -24980.303,E2 -24980.303} C_VEL
LIN {X 0,Y 181.481,Z 443.905,A -85,B 0,C 180,E1 -24981.156,E2 -24981.156} C_VEL
LIN {X 0,Y 183.343,Z 429.982,A -85,B 0,C 180,E1 -24981.785,E2 -24981.785} C_VEL
LIN {X 0,Y 184.97,Z 410.4,A -85,B 0,C 180,E1 -24982.39,E2 -24982.39} C_VEL
LIN {X 0,Y 181.46,Z 400.832,A -85,B 0,C 180,E1 -24984.794,E2 -24984.794} C_VEL
LIN {X 0,Y 177.632,Z 391.83,A -85,B 0,C 180,E1 -24987.632,E2 -24987.632} C_VEL
LIN {X 0,Y 173.885,Z 383.922,A -85,B 0,C 180,E1 -24990.743,E2 -24990.743} C_VEL
LIN {X 0,Y 170.968,Z 378.264,A -85,B 0,C 180,E1 -24993.495,E2 -24993.495} C_VEL
LIN {X 0,Y 168.666,Z 374.102,A -85,B 0,C 180,E1 -24995.957,E2 -24995.957} C_VEL
LIN {X 0,Y 166.456,Z 370.113,A -85,B 0,C 180,E1 -24998.705,E2 -24998.705} C_VEL
LIN {X 0,Y 163.919,Z 366.925,A -85,B 0,C 180,E1 -25002.42,E2 -25002.42} C_VEL
LIN {X 0,Y 163.201,Z 365.4,A -85,B 0,C 180,E1 -25003.826,E2 -25003.826} C_VEL
LIN {X 0,Y 160.842,Z 362.851,A -85,B 0,C 180,E1 -25009.696,E2 -25009.696} C_VEL
LIN {X 0,Y 160.314,Z 360.155,A -85,B 0,C 180,E1 -25014.024,E2 -25014.024} C_VEL
LIN {X 0,Y 160.437,Z 360.155,A -85,B 0,C 180,E1 -25018.712,E2 -25018.712} C_VEL
LIN {X 0,Y 161.085,Z 363.065,A -85,B 0,C 180,E1 -25022.814,E2 -25022.814} C_VEL
LIN {X 0,Y 163.474,Z 365.499,A -85,B 0,C 180,E1 -25028.312,E2 -25028.312} C_VEL
LIN {X 0,Y 165.255,Z 368.787,A -85,B 0,C 180,E1 -25031.367,E2 -25031.367} C_VEL
LIN {X 0,Y 166.764,Z 370.477,A -85,B 0,C 180,E1 -25033.364,E2 -25033.364} C_VEL
LIN {X 0,Y 170.27,Z 375.743,A -85,B 0,C 180,E1 -25037.336,E2 -25037.336} C_VEL
LIN {X 0,Y 173.021,Z 379.956,A -85,B 0,C 180,E1 -25039.937,E2 -25039.937} C_VEL
LIN {X 0,Y 175.943,Z 384.607,A -85,B 0,C 180,E1 -25042.379,E2 -25042.379} C_VEL
LIN {X 0,Y 180.515,Z 392.457,A -85,B 0,C 180,E1 -25045.742,E2 -25045.742} C_VEL
LIN {X 0,Y 185.175,Z 401.462,A -85,B 0,C 180,E1 -25048.77,E2 -25048.77} C_VEL
LIN {X 0,Y 185.6,Z 402.364,A -85,B 0,C 180,E1 -25049.032,E2 -25049.032} C_VEL
LIN {X 0,Y 183.311,Z 426.831,A -85,B 0,C 180,E1 -25049.808,E2 -25049.808} C_VEL
LIN {X 0,Y 181.17,Z 439.888,A -85,B 0,C 180,E1 -25050.595,E2 -25050.595} C_VEL
LIN {X 0,Y 178.096,Z 452.395,A -85,B 0,C 180,E1 -25051.693,E2 -25051.693} C_VEL
LIN {X 0,Y 174.018,Z 464.288,A -85,B 0,C 180,E1 -25053.071,E2 -25053.071} C_VEL
LIN {X 0,Y 169.112,Z 475.979,A -85,B 0,C 180,E1 -25054.944,E2 -25054.944} C_VEL
LIN {X 0,Y 164.375,Z 485.691,A -85,B 0,C 180,E1 -25057.086,E2 -25057.086} C_VEL
LIN {X 0,Y 159.349,Z 494.31,A -85,B 0,C 180,E1 -25059.484,E2 -25059.484} C_VEL
LIN {X 0,Y 153.213,Z 503.354,A -85,B 0,C 180,E1 -25062.785,E2 -25062.785} C_VEL
LIN {X 0,Y 147.634,Z 510.593,A -85,B 0,C 180,E1 -25066.352,E2 -25066.352} C_VEL
LIN {X 0,Y 142.575,Z 516.314,A -85,B 0,C 180,E1 -25070.15,E2 -25070.15} C_VEL
LIN {X 0,Y 137.422,Z 521.428,A -85,B 0,C 180,E1 -25074.914,E2 -25074.914} C_VEL
LIN {X 0,Y 134.394,Z 524.14,A -85,B 0,C 180,E1 -25078.473,E2 -25078.473} C_VEL
LIN {X 0,Y 132.29,Z 525.79,A -85,B 0,C 180,E1 -25081.439,E2 -25081.439} C_VEL
LIN {X 0,Y 130.538,Z 527.028,A -85,B 0,C 180,E1 -25084.49,E2 -25084.49} C_VEL
LIN {X 0,Y 129.036,Z 527.892,A -85,B 0,C 180,E1 -25087.809,E2 -25087.809} C_VEL
LIN {X 0,Y 127.148,Z 528.237,A -85,B 0,C 180,E1 -25093.958,E2 -25093.958} C_VEL
LIN {X 0,Y 126.628,Z 527.845,A -85,B 0,C 180,E1 -25097.175,E2 -25097.175} C_VEL
LIN {X 0,Y 126.452,Z 527.052,A -85,B 0,C 180,E1 -25100.404,E2 -25100.404} C_VEL
LIN {X 0,Y 126.849,Z 524.768,A -85,B 0,C 180,E1 -25105.791,E2 -25105.791} C_VEL
LIN {X 0,Y 127.669,Z 520.943,A -85,B 0,C 180,E1 -25111.579,E2 -25111.579} C_VEL
LIN {X 0,Y 129.165,Z 516.637,A -85,B 0,C 180,E1 -25116.249,E2 -25116.249} C_VEL
LIN {X 0,Y 131.642,Z 510.147,A -85,B 0,C 180,E1 -25121.551,E2 -25121.551} C_VEL
LIN {X 0,Y 134.46,Z 503.025,A -85,B 0,C 180,E1 -25125.929,E2 -25125.929} C_VEL
LIN {X 0,Y 138.003,Z 494.164,A -85,B 0,C 180,E1 -25130.108,E2 -25130.108} C_VEL
LIN {X 0,Y 141.472,Z 485.067,A -85,B 0,C 180,E1 -25133.419,E2 -25133.419} C_VEL
LIN {X 0,Y 144.915,Z 474.971,A -85,B 0,C 180,E1 -25136.268,E2 -25136.268} C_VEL
LIN {X 0,Y 148.23,Z 463.765,A -85,B 0,C 180,E1 -25138.691,E2 -25138.691} C_VEL
LIN {X 0,Y 151.05,Z 451.247,A -85,B 0,C 180,E1 -25140.786,E2 -25140.786} C_VEL
LIN {X 0,Y 153.303,Z 438.974,A -85,B 0,C 180,E1 -25142.206,E2 -25142.206} C_VEL
LIN {X 0,Y 154.995,Z 425.005,A -85,B 0,C 180,E1 -25143.29,E2 -25143.29} C_VEL
LIN {X 0,Y 158.03,Z 377.304,A -85,B 0,C 180,E1 -25145.26,E2 -25145.26} C_VEL
LIN {X 0,Y 153.262,Z 367.165,A -85,B 0,C 180,E1 -25147.43,E2 -25147.43} C_VEL
LIN {X 0,Y 147.137,Z 356.033,A -85,B 0,C 180,E1 -25150.424,E2 -25150.424} C_VEL
LIN {X 0,Y 141.52,Z 347.341,A -85,B 0,C 180,E1 -25153.444,E2 -25153.444} C_VEL
LIN {X 0,Y 138.774,Z 343.449,A -85,B 0,C 180,E1 -25155.051,E2 -25155.051} C_VEL
LIN {X 0,Y 136.453,Z 340.086,A -85,B 0,C 180,E1 -25156.513,E2 -25156.513} C_VEL
LIN {X 0,Y 133.495,Z 336.414,A -85,B 0,C 180,E1 -25158.469,E2 -25158.469} C_VEL
LIN {X 0,Y 132.692,Z 334.831,A -85,B 0,C 180,E1 -25159.084,E2 -25159.084} C_VEL
LIN {X 0,Y 130.276,Z 332.703,A -85,B 0,C 180,E1 -25160.784,E2 -25160.784} C_VEL
LIN {X 0,Y 129.159,Z 330.317,A -85,B 0,C 180,E1 -25161.759,E2 -25161.759} C_VEL
LIN {X 0,Y 128.961,Z 329.416,A -85,B 0,C 180,E1 -25162.062,E2 -25162.062} C_VEL
LIN {X 0,Y 128.977,Z 329.394,A -85,B 0,C 180,E1 -25166.981,E2 -25166.981} C_VEL
LIN {X 0,Y 129.022,Z 329.412,A -85,B 0,C 180,E1 -25170.642,E2 -25170.642} C_VEL
LIN {X 0,Y 129.113,Z 329.388,A -85,B 0,C 180,E1 -25177.601,E2 -25177.601} C_VEL
LIN {X 0,Y 129.153,Z 329.39,A -85,B 0,C 180,E1 -25180.943,E2 -25180.943} C_VEL
LIN {X 0,Y 129.352,Z 329.358,A -85,B 0,C 180,E1 -25187.963,E2 -25187.963} C_VEL
LIN {X 0,Y 129.475,Z 329.355,A -85,B 0,C 180,E1 -25190.627,E2 -25190.627} C_VEL
LIN {X 0,Y 130.072,Z 329.28,A -85,B 0,C 180,E1 -25199.999,E2 -25199.999} C_VEL
LIN {X 0,Y 129.466,Z 329.342,A -85,B 0,C 180,E1 -25209.372,E2 -25209.372} C_VEL
LIN {X 0,Y 129.302,Z 329.376,A -85,B 0,C 180,E1 -25212.556,E2 -25212.556} C_VEL
LIN {X 0,Y 129.089,Z 329.4,A -85,B 0,C 180,E1 -25219.065,E2 -25219.065} C_VEL
LIN {X 0,Y 129.049,Z 329.406,A -85,B 0,C 180,E1 -25222.409,E2 -25222.409} C_VEL
LIN {X 0,Y 129.068,Z 329.427,A -85,B 0,C 180,E1 -25228.453,E2 -25228.453} C_VEL
LIN {X 0,Y 129.887,Z 332.042,A -85,B 0,C 180,E1 -25229.262,E2 -25229.262} C_VEL
LIN {X 0,Y 131.768,Z 334.2,A -85,B 0,C 180,E1 -25230.665,E2 -25230.665} C_VEL
LIN {X 0,Y 132.958,Z 335.082,A -85,B 0,C 180,E1 -25231.465,E2 -25231.465} C_VEL
LIN {X 0,Y 134.984,Z 338.445,A -85,B 0,C 180,E1 -25232.921,E2 -25232.921} C_VEL
LIN {X 0,Y 136.66,Z 340.322,A -85,B 0,C 180,E1 -25233.984,E2 -25233.984} C_VEL
LIN {X 0,Y 139.127,Z 343.773,A -85,B 0,C 180,E1 -25235.515,E2 -25235.515} C_VEL
LIN {X 0,Y 142.904,Z 349.568,A -85,B 0,C 180,E1 -25237.71,E2 -25237.71} C_VEL
LIN {X 0,Y 148.178,Z 360.005,A -85,B 0,C 180,E1 -25240.62,E2 -25240.62} C_VEL
LIN {X 0,Y 153.02,Z 371.581,A -85,B 0,C 180,E1 -25243.13,E2 -25243.13} C_VEL
LIN {X 0,Y 156.198,Z 381.056,A -85,B 0,C 180,E1 -25244.755,E2 -25244.755} C_VEL
LIN {X 0,Y 157.058,Z 396.303,A -85,B 0,C 180,E1 -25245.92,E2 -25245.92} C_VEL
LIN {X 0,Y 154.462,Z 436.823,A -85,B 0,C 180,E1 -25247.624,E2 -25247.624} C_VEL
LIN {X 0,Y 152.722,Z 449.782,A -85,B 0,C 180,E1 -25248.583,E2 -25248.583} C_VEL
LIN {X 0,Y 150.272,Z 462.349,A -85,B 0,C 180,E1 -25249.977,E2 -25249.977} C_VEL
LIN {X 0,Y 147.399,Z 473.517,A -85,B 0,C 180,E1 -25251.693,E2 -25251.693} C_VEL
LIN {X 0,Y 143.814,Z 485.149,A -85,B 0,C 180,E1 -25254.094,E2 -25254.094} C_VEL
LIN {X 0,Y 140.186,Z 495.63,A -85,B 0,C 180,E1 -25256.959,E2 -25256.959} C_VEL
LIN {X 0,Y 137.06,Z 504.205,A -85,B 0,C 180,E1 -25260.001,E2 -25260.001} C_VEL
LIN {X 0,Y 133.941,Z 511.789,A -85,B 0,C 180,E1 -25263.343,E2 -25263.343} C_VEL
LIN {X 0,Y 131.935,Z 517.403,A -85,B 0,C 180,E1 -25266.45,E2 -25266.45} C_VEL
LIN {X 0,Y 129.454,Z 524.081,A -85,B 0,C 180,E1 -25270.988,E2 -25270.988} C_VEL
LIN {X 0,Y 127.712,Z 529.392,A -85,B 0,C 180,E1 -25275.66,E2 -25275.66} C_VEL
LIN {X 0,Y 126.842,Z 533.516,A -85,B 0,C 180,E1 -25280.43,E2 -25280.43} C_VEL
LIN {X 0,Y 126.563,Z 535.651,A -85,B 0,C 180,E1 -25283.622,E2 -25283.622} C_VEL
LIN {X 0,Y 126.62,Z 537.66,A -85,B 0,C 180,E1 -25287.533,E2 -25287.533} C_VEL
LIN {X 0,Y 126.74,Z 538.594,A -85,B 0,C 180,E1 -25289.998,E2 -25289.998} C_VEL
LIN {X 0,Y 126.544,Z 539.42,A -85,B 0,C 180,E1 -25293.182,E2 -25293.182} C_VEL
LIN {X 0,Y 126.533,Z 539.81,A -85,B 0,C 180,E1 -25296.376,E2 -25296.376} C_VEL
LIN {X 0,Y 127.388,Z 539.421,A -85,B 0,C 180,E1 -25302.747,E2 -25302.747} C_VEL
LIN {X 0,Y 128.817,Z 538.211,A -85,B 0,C 180,E1 -25307.077,E2 -25307.077} C_VEL
LIN {X 0,Y 131.459,Z 535.892,A -85,B 0,C 180,E1 -25311.975,E2 -25311.975} C_VEL
LIN {X 0,Y 134.752,Z 532.726,A -85,B 0,C 180,E1 -25316.314,E2 -25316.314} C_VEL
LIN {X 0,Y 137.557,Z 529.831,A -85,B 0,C 180,E1 -25319.266,E2 -25319.266} C_VEL
LIN {X 0,Y 139.078,Z 527.491,A -85,B 0,C 180,E1 -25321.422,E2 -25321.422} C_VEL
LIN {X 0,Y 140.384,Z 523.273,A -85,B 0,C 180,E1 -25325.074,E2 -25325.074} C_VEL
LIN {X 0,Y 142.151,Z 518.489,A -85,B 0,C 180,E1 -25328.509,E2 -25328.509} C_VEL
LIN {X 0,Y 144.298,Z 515.184,A -85,B 0,C 180,E1 -25330.259,E2 -25330.259} C_VEL
LIN {X 0,Y 150.601,Z 506.797,A -85,B 0,C 180,E1 -25333.496,E2 -25333.496} C_VEL
LIN {X 0,Y 156.213,Z 498.096,A -85,B 0,C 180,E1 -25336.039,E2 -25336.039} C_VEL
LIN {X 0,Y 161.665,Z 488.573,A -85,B 0,C 180,E1 -25338.111,E2 -25338.111} C_VEL
LIN {X 0,Y 166.706,Z 478.196,A -85,B 0,C 180,E1 -25339.826,E2 -25339.826} C_VEL
LIN {X 0,Y 171.24,Z 466.824,A -85,B 0,C 180,E1 -25341.239,E2 -25341.239} C_VEL
LIN {X 0,Y 174.844,Z 455.224,A -85,B 0,C 180,E1 -25342.293,E2 -25342.293} C_VEL
LIN {X 0,Y 177.783,Z 442.101,A -85,B 0,C 180,E1 -25343.126,E2 -25343.126} C_VEL
LIN {X 0,Y 179.533,Z 429.089,A -85,B 0,C 180,E1 -25343.676,E2 -25343.676} C_VEL
LIN {X 0,Y 180.894,Z 412.937,A -85,B 0,C 180,E1 -25344.184,E2 -25344.184} C_VEL
LIN {X 0,Y 177.648,Z 403.916,A -85,B 0,C 180,E1 -25346.629,E2 -25346.629} C_VEL
LIN {X 0,Y 174.191,Z 395.653,A -85,B 0,C 180,E1 -25349.449,E2 -25349.449} C_VEL
LIN {X 0,Y 171.192,Z 389.076,A -85,B 0,C 180,E1 -25352.187,E2 -25352.187} C_VEL
LIN {X 0,Y 168.875,Z 384.258,A -85,B 0,C 180,E1 -25354.573,E2 -25354.573} C_VEL
LIN {X 0,Y 166.848,Z 380.384,A -85,B 0,C 180,E1 -25356.908,E2 -25356.908} C_VEL
LIN {X 0,Y 165.042,Z 376.872,A -85,B 0,C 180,E1 -25359.32,E2 -25359.32} C_VEL
LIN {X 0,Y 162.587,Z 373.574,A -85,B 0,C 180,E1 -25363.158,E2 -25363.158} C_VEL
LIN {X 0,Y 161.981,Z 372.248,A -85,B 0,C 180,E1 -25364.428,E2 -25364.428} C_VEL
LIN {X 0,Y 159.854,Z 369.742,A -85,B 0,C 180,E1 -25370.147,E2 -25370.147} C_VEL
LIN {X 0,Y 159.43,Z 367.349,A -85,B 0,C 180,E1 -25373.991,E2 -25373.991} C_VEL
LIN {X 0,Y 159.518,Z 367.259,A -85,B 0,C 180,E1 -25378.406,E2 -25378.406} C_VEL
LIN {X 0,Y 160.117,Z 370.05,A -85,B 0,C 180,E1 -25382.516,E2 -25382.516} C_VEL
LIN {X 0,Y 162.254,Z 372.405,A -85,B 0,C 180,E1 -25387.748,E2 -25387.748} C_VEL
LIN {X 0,Y 164.153,Z 375.81,A -85,B 0,C 180,E1 -25391.112,E2 -25391.112} C_VEL
LIN {X 0,Y 165.375,Z 377.372,A -85,B 0,C 180,E1 -25392.814,E2 -25392.814} C_VEL
LIN {X 0,Y 168.418,Z 382.097,A -85,B 0,C 180,E1 -25396.458,E2 -25396.458} C_VEL
LIN {X 0,Y 171.133,Z 386.468,A -85,B 0,C 180,E1 -25399.181,E2 -25399.181} C_VEL
LIN {X 0,Y 174.792,Z 392.643,A -85,B 0,C 180,E1 -25402.353,E2 -25402.353} C_VEL
LIN {X 0,Y 179.249,Z 400.861,A -85,B 0,C 180,E1 -25405.705,E2 -25405.705} C_VEL
LIN {X 0,Y 181.468,Z 405.457,A -85,B 0,C 180,E1 -25407.235,E2 -25407.235} C_VEL
LIN {X 0,Y 179.347,Z 427.462,A -85,B 0,C 180,E1 -25407.962,E2 -25407.962} C_VEL
LIN {X 0,Y 177.107,Z 440.498,A -85,B 0,C 180,E1 -25408.748,E2 -25408.748} C_VEL
LIN {X 0,Y 174.097,Z 452.368,A -85,B 0,C 180,E1 -25409.785,E2 -25409.785} C_VEL
LIN {X 0,Y 170.192,Z 463.531,A -85,B 0,C 180,E1 -25411.037,E2 -25411.037} C_VEL
LIN {X 0,Y 165.83,Z 473.85,A -85,B 0,C 180,E1 -25412.617,E2 -25412.617} C_VEL
LIN {X 0,Y 161.241,Z 483.182,A -85,B 0,C 180,E1 -25414.517,E2 -25414.517} C_VEL
LIN {X 0,Y 155.972,Z 492.298,A -85,B 0,C 180,E1 -25416.891,E2 -25416.891} C_VEL
LIN {X 0,Y 150.472,Z 500.402,A -85,B 0,C 180,E1 -25419.59,E2 -25419.59} C_VEL
LIN {X 0,Y 144.349,Z 508.296,A -85,B 0,C 180,E1 -25423.09,E2 -25423.09} C_VEL
LIN {X 0,Y 138.803,Z 514.555,A -85,B 0,C 180,E1 -25426.881,E2 -25426.881} C_VEL
LIN {X 0,Y 133.829,Z 519.496,A -85,B 0,C 180,E1 -25430.939,E2 -25430.939} C_VEL
LIN {X 0,Y 129.518,Z 523.276,A -85,B 0,C 180,E1 -25435.269,E2 -25435.269} C_VEL
LIN {X 0,Y 125.957,Z 526.001,A -85,B 0,C 180,E1 -25439.859,E2 -25439.859} C_VEL
LIN {X 0,Y 122.444,Z 528.133,A -85,B 0,C 180,E1 -25446.312,E2 -25446.312} C_VEL
LIN {X 0,Y 121.176,Z 528.565,A -85,B 0,C 180,E1 -25449.638,E2 -25449.638} C_VEL
LIN {X 0,Y 120.249,Z 528.585,A -85,B 0,C 180,E1 -25453.011,E2 -25453.011} C_VEL
LIN {X 0,Y 119.369,Z 527.467,A -85,B 0,C 180,E1 -25459.829,E2 -25459.829} C_VEL
LIN {X 0,Y 119.774,Z 525.021,A -85,B 0,C 180,E1 -25465.975,E2 -25465.975} C_VEL
LIN {X 0,Y 120.585,Z 521.484,A -85,B 0,C 180,E1 -25471.672,E2 -25471.672} C_VEL
LIN {X 0,Y 122.099,Z 517.243,A -85,B 0,C 180,E1 -25476.613,E2 -25476.613} C_VEL
LIN {X 0,Y 124.729,Z 510.826,A -85,B 0,C 180,E1 -25482.2,E2 -25482.2} C_VEL
LIN {X 0,Y 127.666,Z 503.815,A -85,B 0,C 180,E1 -25486.801,E2 -25486.801} C_VEL
LIN {X 0,Y 131.393,Z 495.045,A -85,B 0,C 180,E1 -25491.166,E2 -25491.166} C_VEL
LIN {X 0,Y 135.398,Z 485.079,A -85,B 0,C 180,E1 -25494.946,E2 -25494.946} C_VEL
LIN {X 0,Y 139.046,Z 474.888,A -85,B 0,C 180,E1 -25497.876,E2 -25497.876} C_VEL
LIN {X 0,Y 142.519,Z 463.594,A -85,B 0,C 180,E1 -25500.364,E2 -25500.364} C_VEL
LIN {X 0,Y 145.283,Z 451.939,A -85,B 0,C 180,E1 -25502.356,E2 -25502.356} C_VEL
LIN {X 0,Y 147.732,Z 439.104,A -85,B 0,C 180,E1 -25503.885,E2 -25503.885} C_VEL
LIN {X 0,Y 149.435,Z 425.9,A -85,B 0,C 180,E1 -25504.93,E2 -25504.93} C_VEL
LIN {X 0,Y 151.521,Z 395.781,A -85,B 0,C 180,E1 -25506.234,E2 -25506.234} C_VEL
LIN {X 0,Y 152.568,Z 379.613,A -85,B 0,C 180,E1 -25506.889,E2 -25506.889} C_VEL
LIN {X 0,Y 148.391,Z 370.614,A -85,B 0,C 180,E1 -25508.956,E2 -25508.956} C_VEL
LIN {X 0,Y 142.832,Z 360.314,A -85,B 0,C 180,E1 -25511.902,E2 -25511.902} C_VEL
LIN {X 0,Y 135.969,Z 349.599,A -85,B 0,C 180,E1 -25515.977,E2 -25515.977} C_VEL
LIN {X 0,Y 132.386,Z 344.76,A -85,B 0,C 180,E1 -25518.366,E2 -25518.366} C_VEL
LIN {X 0,Y 129.962,Z 341.203,A -85,B 0,C 180,E1 -25520.169,E2 -25520.169} C_VEL
LIN {X 0,Y 127.198,Z 338.113,A -85,B 0,C 180,E1 -25522.32,E2 -25522.32} C_VEL
LIN {X 0,Y 125.972,Z 335.86,A -85,B 0,C 180,E1 -25523.443,E2 -25523.443} C_VEL
LIN {X 0,Y 123.427,Z 333.859,A -85,B 0,C 180,E1 -25525.661,E2 -25525.661} C_VEL
LIN {X 0,Y 122.197,Z 331.453,A -85,B 0,C 180,E1 -25527.003,E2 -25527.003} C_VEL
LIN {X 0,Y 121.914,Z 330.277,A -85,B 0,C 180,E1 -25527.53,E2 -25527.53} C_VEL
LIN {X 0,Y 121.941,Z 330.27,A -85,B 0,C 180,E1 -25532.542,E2 -25532.542} C_VEL
LIN {X 0,Y 122.032,Z 330.262,A -85,B 0,C 180,E1 -25537.146,E2 -25537.146} C_VEL
LIN {X 0,Y 122.102,Z 330.241,A -85,B 0,C 180,E1 -25543.273,E2 -25543.273} C_VEL
LIN {X 0,Y 122.402,Z 330.238,A -85,B 0,C 180,E1 -25550.08,E2 -25550.08} C_VEL
LIN {X 0,Y 122.563,Z 330.18,A -85,B 0,C 180,E1 -25556.712,E2 -25556.712} C_VEL
LIN {X 0,Y 123.025,Z 330.157,A -85,B 0,C 180,E1 -25559.999,E2 -25559.999} C_VEL
LIN {X 0,Y 122.408,Z 330.197,A -85,B 0,C 180,E1 -25566.593,E2 -25566.593} C_VEL
LIN {X 0,Y 122.395,Z 330.228,A -85,B 0,C 180,E1 -25569.919,E2 -25569.919} C_VEL
LIN {X 0,Y 122.192,Z 330.258,A -85,B 0,C 180,E1 -25573.3,E2 -25573.3} C_VEL
LIN {X 0,Y 121.994,Z 330.29,A -85,B 0,C 180,E1 -25580.221,E2 -25580.221} C_VEL
LIN {X 0,Y 121.976,Z 330.355,A -85,B 0,C 180,E1 -25583.03,E2 -25583.03} C_VEL
LIN {X 0,Y 122.713,Z 332.78,A -85,B 0,C 180,E1 -25583.97,E2 -25583.97} C_VEL
LIN {X 0,Y 124.527,Z 334.943,A -85,B 0,C 180,E1 -25585.712,E2 -25585.712} C_VEL
LIN {X 0,Y 126.262,Z 336.119,A -85,B 0,C 180,E1 -25587.159,E2 -25587.159} C_VEL
LIN {X 0,Y 128.017,Z 339.215,A -85,B 0,C 180,E1 -25588.72,E2 -25588.72} C_VEL
LIN {X 0,Y 130.151,Z 341.353,A -85,B 0,C 180,E1 -25590.329,E2 -25590.329} C_VEL
LIN {X 0,Y 132.578,Z 344.912,A -85,B 0,C 180,E1 -25592.124,E2 -25592.124} C_VEL
LIN {X 0,Y 136.605,Z 350.613,A -85,B 0,C 180,E1 -25594.802,E2 -25594.802} C_VEL
LIN {X 0,Y 139.426,Z 355.122,A -85,B 0,C 180,E1 -25596.543,E2 -25596.543} C_VEL
LIN {X 0,Y 144.344,Z 365.428,A -85,B 0,C 180,E1 -25599.466,E2 -25599.466} C_VEL
LIN {X 0,Y 148.669,Z 376.342,A -85,B 0,C 180,E1 -25601.891,E2 -25601.891} C_VEL
LIN {X 0,Y 150.924,Z 383.408,A -85,B 0,C 180,E1 -25603.152,E2 -25603.152} C_VEL
LIN {X 0,Y 151.612,Z 397.555,A -85,B 0,C 180,E1 -25604.272,E2 -25604.272} C_VEL
LIN {X 0,Y 149.016,Z 435.697,A -85,B 0,C 180,E1 -25605.877,E2 -25605.877} C_VEL
LIN {X 0,Y 147.229,Z 448.974,A -85,B 0,C 180,E1 -25606.867,E2 -25606.867} C_VEL
LIN {X 0,Y 144.641,Z 461.849,A -85,B 0,C 180,E1 -25608.31,E2 -25608.31} C_VEL
LIN {X 0,Y 141.391,Z 473.858,A -85,B 0,C 180,E1 -25610.208,E2 -25610.208} C_VEL
LIN {X 0,Y 137.65,Z 485.367,A -85,B 0,C 180,E1 -25612.675,E2 -25612.675} C_VEL
LIN {X 0,Y 133.851,Z 495.747,A -85,B 0,C 180,E1 -25615.634,E2 -25615.634} C_VEL
LIN {X 0,Y 130.216,Z 505.069,A -85,B 0,C 180,E1 -25619.152,E2 -25619.152} C_VEL
LIN {X 0,Y 126.879,Z 512.994,A -85,B 0,C 180,E1 -25622.97,E2 -25622.97} C_VEL
LIN {X 0,Y 123.997,Z 520.274,A -85,B 0,C 180,E1 -25627.504,E2 -25627.504} C_VEL
LIN {X 0,Y 121.306,Z 527.187,A -85,B 0,C 180,E1 -25633.159,E2 -25633.159} C_VEL
LIN {X 0,Y 120.049,Z 531.745,A -85,B 0,C 180,E1 -25638.174,E2 -25638.174} C_VEL
LIN {X 0,Y 119.484,Z 535.191,A -85,B 0,C 180,E1 -25643.242,E2 -25643.242} C_VEL
LIN {X 0,Y 119.553,Z 537.462,A -85,B 0,C 180,E1 -25647.933,E2 -25647.933} C_VEL
LIN {X 0,Y 119.521,Z 538.635,A -85,B 0,C 180,E1 -25651.583,E2 -25651.583} C_VEL
LIN {X 0,Y 119.455,Z 539.466,A -85,B 0,C 180,E1 -25656.755,E2 -25656.755} C_VEL
LIN {X 0,Y 120.453,Z 539.124,A -85,B 0,C 180,E1 -25663.494,E2 -25663.494} C_VEL
LIN {X 0,Y 122.946,Z 537.256,A -85,B 0,C 180,E1 -25670.056,E2 -25670.056} C_VEL
LIN {X 0,Y 124.887,Z 535.69,A -85,B 0,C 180,E1 -25673.197,E2 -25673.197} C_VEL
LIN {X 0,Y 128.416,Z 532.574,A -85,B 0,C 180,E1 -25677.72,E2 -25677.72} C_VEL
LIN {X 0,Y 132.789,Z 528.26,A -85,B 0,C 180,E1 -25682.134,E2 -25682.134} C_VEL
LIN {X 0,Y 138.446,Z 522.117,A -85,B 0,C 180,E1 -25686.615,E2 -25686.615} C_VEL
LIN {X 0,Y 144.298,Z 515.184,A -85,B 0,C 180,E1 -25690.259,E2 -25690.259} C_VEL
LIN {X 0,Y 146.528,Z 511.686,A -85,B 0,C 180,E1 -25691.911,E2 -25691.911} C_VEL
LIN {X 0,Y 148.904,Z 505.656,A -85,B 0,C 180,E1 -25694.823,E2 -25694.823} C_VEL
LIN {X 0,Y 151.396,Z 499.175,A -85,B 0,C 180,E1 -25697.516,E2 -25697.516} C_VEL
LIN {X 0,Y 153.654,Z 494.853,A -85,B 0,C 180,E1 -25698.768,E2 -25698.768} C_VEL
LIN {X 0,Y 158.995,Z 485.375,A -85,B 0,C 180,E1 -25700.671,E2 -25700.671} C_VEL
LIN {X 0,Y 164.171,Z 474.252,A -85,B 0,C 180,E1 -25702.367,E2 -25702.367} C_VEL
LIN {X 0,Y 168.933,Z 461.774,A -85,B 0,C 180,E1 -25703.709,E2 -25703.709} C_VEL
LIN {X 0,Y 172.492,Z 449.117,A -85,B 0,C 180,E1 -25704.69,E2 -25704.69} C_VEL
LIN {X 0,Y 174.872,Z 436.625,A -85,B 0,C 180,E1 -25705.358,E2 -25705.358} C_VEL
LIN {X 0,Y 177.037,Z 415.684,A -85,B 0,C 180,E1 -25706.03,E2 -25706.03} C_VEL
LIN {X 0,Y 173.883,Z 406.699,A -85,B 0,C 180,E1 -25708.66,E2 -25708.66} C_VEL
LIN {X 0,Y 170.395,Z 398.185,A -85,B 0,C 180,E1 -25711.862,E2 -25711.862} C_VEL
LIN {X 0,Y 167.199,Z 390.988,A -85,B 0,C 180,E1 -25715.265,E2 -25715.265} C_VEL
LIN {X 0,Y 165.041,Z 386.59,A -85,B 0,C 180,E1 -25717.93,E2 -25717.93} C_VEL
LIN {X 0,Y 163.459,Z 383.411,A -85,B 0,C 180,E1 -25720.215,E2 -25720.215} C_VEL
LIN {X 0,Y 161.226,Z 380.096,A -85,B 0,C 180,E1 -25724.028,E2 -25724.028} C_VEL
LIN {X 0,Y 160.769,Z 379.083,A -85,B 0,C 180,E1 -25725.063,E2 -25725.063} C_VEL
LIN {X 0,Y 158.845,Z 376.587,A -85,B 0,C 180,E1 -25730.752,E2 -25730.752} C_VEL
LIN {X 0,Y 158.531,Z 374.333,A -85,B 0,C 180,E1 -25734.436,E2 -25734.436} C_VEL
LIN {X 0,Y 158.605,Z 374.232,A -85,B 0,C 180,E1 -25737.957,E2 -25737.957} C_VEL
LIN {X 0,Y 159.112,Z 376.961,A -85,B 0,C 180,E1 -25742.057,E2 -25742.057} C_VEL
LIN {X 0,Y 161.048,Z 379.292,A -85,B 0,C 180,E1 -25747.169,E2 -25747.169} C_VEL
LIN {X 0,Y 163.135,Z 382.945,A -85,B 0,C 180,E1 -25750.977,E2 -25750.977} C_VEL
LIN {X 0,Y 164.235,Z 384.698,A -85,B 0,C 180,E1 -25752.591,E2 -25752.591} C_VEL
LIN {X 0,Y 166.824,Z 388.839,A -85,B 0,C 180,E1 -25755.815,E2 -25755.815} C_VEL
LIN {X 0,Y 169.832,Z 393.841,A -85,B 0,C 180,E1 -25758.942,E2 -25758.942} C_VEL
LIN {X 0,Y 174.014,Z 401.492,A -85,B 0,C 180,E1 -25762.641,E2 -25762.641} C_VEL
LIN {X 0,Y 177.581,Z 408.802,A -85,B 0,C 180,E1 -25765.406,E2 -25765.406} C_VEL
LIN {X 0,Y 175.525,Z 428.519,A -85,B 0,C 180,E1 -25766.053,E2 -25766.053} C_VEL
LIN {X 0,Y 173.236,Z 441.117,A -85,B 0,C 180,E1 -25766.812,E2 -25766.812} C_VEL
